(***********************************************************************************************)
(* HMI Alarme*)
(***********************************************************************************************)
FOR idx := 1 TO 500 BY 1 DO
    HMI.xArAlarmHMI[idx] := HMI.strArALARM[idx].xAlarmOUT;
END_FOR

FOR idx := 1 TO 100 BY 1 DO
    HMI.xArAlarmHMI[idx + 5000] := HMI.strArMSG[idx].xAlarmOUT;
END_FOR

(***********************************************************************************************)
(* Cycle Time *)
(***********************************************************************************************)
_FB_SystemTime(timeLoDW => dw_ActTime, timeHiDW =>);
dw_ActTime := dw_ActTime AND 16#FFFF0000;

IF HMI.btArMain[8].rtrig THEN
    HMI.PieceDoneTmp := 0;
END_IF

(***********************************************************************************************)
(* Operating hours  *)
(***********************************************************************************************)
(* 0.5' Blinker *)
BLINK_500(IN := NOT BLINK_500_.Q, PT := T#500MS, Q => x_BLINK_500);
BLINK_500_(IN := NOT BLINK_500.Q, PT := T#500MS);
(* 0.1' Blinker *)
BLINK_100(IN := NOT BLINK_100_.Q, PT := T#100MS, Q => x_BLINK_100);
BLINK_100_(IN := NOT BLINK_100.Q, PT := T#100MS);
(* 6' Ticker *)
TICK6M(IN := NOT TICK6M_.Q, PT := T#1MS, Q => x_TICK6M);
TICK6M_(IN := NOT TICK6M.Q, PT := t#6m);

(* Operating hours *)
IF TICK6M.Q THEN
    (* AUTO *)
    IF (HMI.enState = enState.StateAUTO) THEN
        PERS.udiCount6Mauto := PERS.udiCount6Mauto + 1;
        IF (PERS.udiCount6Mauto >= 10) THEN
            PERS.udiCount6Mauto := 0;
            PERS.udiCountHauto  := PERS.udiCountHauto + 1;
            IF (PERS.udiCountHauto < 0) THEN
                PERS.udiCountHauto := 0;
            END_IF;
        END_IF;
    END_IF;

    (* TOTAL *)
    PERS.udiCount6Mon := PERS.udiCount6Mon + 1;
    IF (PERS.udiCount6Mon >= 10) THEN
        PERS.udiCount6Mon := 0;
        PERS.udiCountHon  := PERS.udiCountHon + 1;
        IF (PERS.udiCountHon < 0) THEN
            PERS.udiCountHon := 0;
        END_IF;
    END_IF;

    //6h
    iCount6h := iCount6h + 1;
END_IF;

//Alarmlog schreiben nach 6h oder bei NOT-AUS
//rtNOTAUS(CLK:=_02_SAFETY.xOUT_ESout);
IF (iCount6h >= 60) OR rtNOTAUS.Q THEN
    iCount6h        := 0;
    HMI.xWriteALlog := NOT HMI.xWriteALlog;
END_IF;

END_PROGRAM

// ---- POUs/10_HMI/_14_STATE.TcPOU
PROGRAM _14_STATE
(****************************************************************************)
//STATE PROGRAMM
//	- Control Buttons
//	- Status Anlage
//
//	05.09.2019/Dj
//
//	Version:
(****************************************************************************)
VAR
    fb_State  : FB_State; //Status der Maschine
    sStateDbg : STRING;   // enState but in string format

    //Control Buttons
    _FB_btAUTO          : FB_BUTTON;
    _FB_btSTEP          : FB_BUTTON;
    _FB_btEND           : FB_BUTTON;
    _FB_btMANU          : FB_BUTTON;
    _FB_btINIT          : FB_BUTTON;
    _FB_btSTOP          : FB_BUTTON;
    _FB_btLEER          : FB_BUTTON;
    _FB_btQUIT          : FB_BUTTON;
    _FB_btSTART         : FB_BUTTON;
    _FB_btRESET_COUNTER : FB_BUTTON;
END_VAR

//****************************************************************************
// 	CONTROL BUTTONS
//****************************************************************************
//	AUTO 
_FB_btAUTO(pbtIN  := ADR(HMI.btArMain[0]),
           xINdis := (HMI.enState < enState.StateREADY),
           xINon  := (HMI.enState = enState.StateAUTO),
           xINerr := FALSE);

//STEP
_FB_btSTEP(pbtIN  := ADR(HMI.btArMain[1]),
           xINdis := (HMI.enState < enState.StateREADY),
           xINon  := (HMI.enState = enState.StateSTEP),
           xINerr := FALSE);

//END
_FB_btEND(pbtIN  := ADR(HMI.btArMain[2]),
          xINdis := (HMI.enState < enState.StateREADY),
          xINon  := (HMI.enState = enState.StateEND),
          xINerr := FALSE);

//MANU
_FB_btMANU(pbtIN  := ADR(HMI.btArMain[3]),
           xINdis := (HMI.enState > enState.StateSTEP) OR
                     (HMI.enState = enState.StateALARM) OR
                     (HMI.enState < enState.StateAIRon),
           xINon  := (HMI.enState = enState.StateMANU),
           xINerr := FALSE);

//INIT
_FB_btINIT(pbtIN  := ADR(HMI.btArMain[4]),
           xINdis := (HMI.enState < enState.StateENGIZED),
           xINon  := (HMI.enState = enState.StateINIT),
           xINerr := FALSE);

//STOP
_FB_btSTOP(pbtIN  := ADR(HMI.btArMain[5]),
           xINdis := (HMI.enState < enState.StateENGIZED),
           xINon  := FALSE,
           xINerr := FALSE);

//LEERFAHREN
_FB_btLEER(pbtIN  := ADR(HMI.btArMain[6]),
           xINdis := FALSE,
           xINon  := FALSE,
           xINerr := FALSE);

//QUIT
_FB_btQUIT(pbtIN  := ADR(HMI.btArMain[7]),
           xINdis := FALSE,
           xINon  := FALSE,
           xINerr := HMI.xAlarm);

_FB_btRESET_COUNTER(pbtIN  := ADR(HMI.btArMain[8]),
                    xINdis := FALSE,
                    xINon  := HMI.btArMain[8].press,
                    xINerr := FALSE);

//START
_FB_btSTART(pbtIN  := ADR(HMI.btArMain[9]),
            xINdis := HMI.enState < enState.StateREADY,
            xINon  := HMI.btArMain[9].on,
            xINerr := FALSE);

//****************************************************************************
// 	STATE FB
//****************************************************************************
fb_State(xIN_AutoInit   := FALSE,
         xIN_DoRef      := FALSE,
         xIN_ENERGIE    := _02_SAFETY.xOUT_MonOut,
         xIN_AIR        := IN.I004_druckwachter_luftdruck_ok,
         xIN_EINRICHTEN := _02_SAFETY.xOUT_Einrichten,
         xIN_AUTO       := HMI.btArMain[0].rtrig,
         xIN_STEP       := HMI.btArMain[1].rtrig,
         xIN_CYCLE      := HMI.btArMain[2].rtrig,
         xIN_MANU       := HMI.btArMain[3].rtrig,
         xIN_INIT       := HMI.btArMain[4].rtrig,
         xIN_STOP       := HMI.btArMain[5].rtrig,
         xIN_LEER       := HMI.btArMain[6].rtrig,
         xIN_InitEND    := (GVL.st105_aut.xOUT_InitDone) AND
                           (GVL.st110_aut.xOUT_InitDone) AND
                           (GVL.st115_aut.xOUT_InitDone) AND
                           (GVL.st120_aut.xOUT_InitDone) AND
                           (GVL.st125_aut.xOUT_InitDone) AND
                           (GVL.st130_aut.xOUT_InitDone) AND
                           (GVL.st135_aut.xOUT_InitDone) AND
                           (GVL.st140_aut.xOUT_InitDone) AND
                           (GVL.st145_aut.xOUT_InitDone) AND
                           (GVL.st150_aut.xOUT_InitDone) AND
                           (GVL.st155_aut.xOUT_InitDone) AND
                           (GVL.st160_aut.xOUT_InitDone) AND
                           (GVL.st165_aut.xOUT_InitDone) AND
                           (GVL.st170_aut.xOUT_InitDone) AND
                           (GVL.st175_aut.xOUT_InitDone) AND
                           (GVL.st176_aut.xOUT_InitDone) AND
                           (GVL.st180_aut.xOUT_InitDone) AND
                           (GVL.st185_aut.xOUT_InitDone),
         xIN_ALARM := MAIN.MoverMan.xOUT_Error OR
                      ((GVL.st105_aut.xOUT_AlarmST) OR
                      (GVL.st110_aut.xOUT_AlarmST) OR
                      (GVL.st115_aut.xOUT_AlarmST) OR
                      (GVL.st120_aut.xOUT_AlarmST) OR
                      (GVL.st125_aut.xOUT_AlarmST) OR
                      (GVL.st128_aut.xOUT_AlarmST) OR
                      (GVL.st130_aut.xOUT_AlarmST) OR
                      (GVL.st135_aut.xOUT_AlarmST) OR
                      (GVL.st140_aut.xOUT_AlarmST) OR
                      (GVL.st145_aut.xOUT_AlarmST) OR
                      (GVL.st150_aut.xOUT_AlarmST) OR
                      (GVL.st155_aut.xOUT_AlarmST) OR
                      (GVL.st160_aut.xOUT_AlarmST) OR
                      (GVL.st165_aut.xOUT_AlarmST) OR
                      (GVL.st170_aut.xOUT_AlarmST) OR
                      (GVL.st175_aut.xOUT_AlarmST) OR
                      (GVL.st180_aut.xOUT_AlarmST) OR
                      (GVL.st185_aut.xOUT_AlarmST)) AND
                      (GVL.st105_aut.xOUT_ErrFlag OR GVL.st105_aut.xOUT_Wait) AND
                      (GVL.st110_aut.xOUT_ErrFlag OR GVL.st110_aut.xOUT_Wait) AND
                      (GVL.st115_aut.xOUT_ErrFlag OR GVL.st115_aut.xOUT_Wait) AND
                      (GVL.st120_aut.xOUT_ErrFlag OR GVL.st120_aut.xOUT_Wait) AND
                      (GVL.st125_aut.xOUT_ErrFlag OR GVL.st125_aut.xOUT_Wait) AND
                      // we ignore the state of ST128
                      (GVL.st130_aut.xOUT_ErrFlag OR GVL.st130_aut.xOUT_Wait) AND
                      (GVL.st135_aut.xOUT_ErrFlag OR GVL.st135_aut.xOUT_Wait) AND
                      // we ignore the state of ST140
                      (GVL.st145_aut.xOUT_ErrFlag OR GVL.st145_aut.xOUT_Wait) AND
                      (GVL.st150_aut.xOUT_ErrFlag OR GVL.st150_aut.xOUT_Wait) AND
                      (GVL.st155_aut.xOUT_ErrFlag OR GVL.st155_aut.xOUT_Wait) AND
                      (GVL.st160_aut.xOUT_ErrFlag OR GVL.st160_aut.xOUT_Wait) AND
                      (GVL.st165_aut.xOUT_ErrFlag OR GVL.st165_aut.xOUT_Wait) AND
                      (GVL.st170_aut.xOUT_ErrFlag OR GVL.st170_aut.xOUT_Wait) AND
                      (GVL.st175_aut.xOUT_ErrFlag OR GVL.st175_aut.xOUT_Wait) AND
                      (GVL.st180_aut.xOUT_ErrFlag OR GVL.st180_aut.xOUT_Wait) AND
                      (GVL.st185_aut.xOUT_ErrFlag OR GVL.st185_aut.xOUT_Wait),
         xIN_LastDone := (NOT (HMI.enState = enState.StateLEER) OR
                         (MAIN.MoverMan.xOUT_AllMoverEmpty AND GVL.st185_aut.xOUT_Done)) AND
                         GVL.st105_aut.xOUT_Wait AND
                         GVL.st110_aut.xOUT_Wait AND
                         GVL.st115_aut.xOUT_Wait AND
                         GVL.st120_aut.xOUT_Wait AND
                         GVL.st125_aut.xOUT_Wait AND
                         GVL.st128_aut.xOUT_Wait AND
                         GVL.st130_aut.xOUT_Wait AND
                         GVL.st135_aut.xOUT_Wait AND
                         GVL.st140_aut.xOUT_Wait AND
                         GVL.st145_aut.xOUT_Wait AND
                         GVL.st150_aut.xOUT_Wait AND
                         GVL.st155_aut.xOUT_Wait AND
                         GVL.st160_aut.xOUT_Wait AND
                         GVL.st165_aut.xOUT_Wait AND
                         GVL.st170_aut.xOUT_Wait AND
                         GVL.st175_aut.xOUT_Wait AND
                         GVL.st180_aut.xOUT_Wait AND
                         GVL.st185_aut.xOUT_Wait,
         xIN_WaitFBs := GVL.st105_aut.xOUT_Wait AND
                        GVL.st110_aut.xOUT_Wait AND
                        GVL.st115_aut.xOUT_Wait AND
                        GVL.st120_aut.xOUT_Wait AND
                        GVL.st125_aut.xOUT_Wait AND
                        GVL.st128_aut.xOUT_Wait AND
                        GVL.st130_aut.xOUT_Wait AND
                        GVL.st135_aut.xOUT_Wait AND
                        GVL.st140_aut.xOUT_Wait AND
                        GVL.st145_aut.xOUT_Wait AND
                        GVL.st150_aut.xOUT_Wait AND
                        GVL.st155_aut.xOUT_Wait AND
                        GVL.st160_aut.xOUT_Wait AND
                        GVL.st165_aut.xOUT_Wait AND
                        GVL.st170_aut.xOUT_Wait AND
                        GVL.st175_aut.xOUT_Wait AND
                        GVL.st180_aut.xOUT_Wait AND
                        GVL.st185_aut.xOUT_Wait,
         enINOUT_State := HMI.enState);

sStateDbg := TO_STRING(HMI.enState);

END_PROGRAM

// ---- POUs/20_AUTO/ST175/Trumpf/TruMark_SingleCmds.TcPOU
PROGRAM TruMark_SingleCmds
(*
	TRUMPF Laser Marking Systems
	============================
	created: 11.01.2019 Erik Haller
	
     +============+
     |SingleCmds  |
     +============+
          |
          v
       +--+------+
       |Input    |	 Interface
       |  -----  |   if_TruMark
       |Output   |
       |  -----  |
       +---------+
               ^
               |
    +==================+
    |TruMark_Ethercat  |
    +==================+
	
	Software Disclaimer:
	THIS SOFTWARE IS PROVIDED "AS IS" AND ANY EXPRESSED OR IMPLIED WARRANTIES, INCLUDING, BUT NOT LIMITED TO,
	THE IMPLIED WARRANTIES OF MERCHANTABILITY AND FITNESS FOR A PARTICULAR PURPOSE ARE DISCLAIMED. 
	IN NO EVENT SHALL THE REGENTS OR CONTRIBUTORS BE LIABLE FOR ANY DIRECT, INDIRECT, INCIDENTAL, SPECIAL, EXEMPLARY, 
	OR CONSEQUENTIAL DAMAGES (INCLUDING, BUT NOT LIMITED TO, PROCUREMENT OF SUBSTITUTE GOODS OR SERVICES; LOSS OF USE, DATA, OR PROFITS;
	OR BUSINESS INTERRUPTION) HOWEVER CAUSED AND ON ANY THEORY OF LIABILITY, WHETHER IN CONTRACT, STRICT LIABILITY, OR TORT (INCLUDING NEGLIGENCE OR OTHERWISE) 
	ARISING IN ANY WAY OUT OF THE USE OF THIS SOFTWARE, EVEN IF ADVISED OF THE POSSIBILITY OF SUCH DAMAGE.
*)



VAR
	iStep : INT;
	abB1 : ARRAY [0..7] OF BOOL;	// used for TLV request 20261
	abB2 : ARRAY [0..7] OF BOOL;	// used for TLV request 20261
	iBitNo : INT;
	sFileName : STRING;
	sVar : STRING;
END_VAR

IF if_TruMark.bError THEN
	iStep := 0;
END_IF

CASE iStep OF
	0: 		// Initialisation
		IF NOT if_TruMark.bError AND NOT if_TruMark.bBusy THEN
			if_SingleCmds.bReady := TRUE;
			iStep := 5;
		END_IF
	
	5:		
		// ---------------------------------------------------------
		// TruMark_Ethercat is Ready --> SELECT Step-No
		// ---------------------------------------------------------
		
		IF if_SingleCmds.bStart THEN
			if_SingleCmds.bStart := FALSE;
			if_SingleCmds.bReady := FALSE;
			iStep := if_SingleCmds.iStepNr;
		END_IF
	
// ============================================================================================================================
// 			T L V   C O M M A N D S		iStep: 10 - 100
// ============================================================================================================================
		
	10:		// -----------------------------------------------------------
			// TLV - Activate Laser / Open Shutter				Attention! Not all Marking Laser have a Shutter
			// -----------------------------------------------------------
		IF NOT if_TruMark.bBusy THEN
			if_TruMark.diTlvTag := 20201;
			if_TruMark.sTlvValueIn := '1';
			if_TruMark.bTlvCmd := TRUE;	
		ELSE
			iStep := 11;
		END_IF
	11:		// Wait for response
		IF NOT if_TruMark.bBusy AND if_TruMark.Status.b0_Laser_On (*AND if_TruMark.Status.b1_Laser_Ready AND if_TruMark.Status.b3_Shutter_Open *) THEN
			iStep := 0;
		END_IF
		
	12:		// -----------------------------------------------------------
			// TLV - Deactivate Laser / Close Shutter				Attention! Not all Marking Laser have a Shutter
			// -----------------------------------------------------------
		IF NOT if_TruMark.bBusy THEN
			if_TruMark.diTlvTag := 20201;
			if_TruMark.sTlvValueIn := '0';
			if_TruMark.bTlvCmd := TRUE;
		ELSE
			iStep := 13;
		END_IF
	13:		// Wait for response
		IF NOT if_TruMark.bBusy AND NOT if_TruMark.Status.b0_Laser_On AND NOT if_TruMark.Status.b1_Laser_Ready (* AND NOT if_TruMark.Status.b3_Shutter_Open *) THEN
			iStep := 0;
		END_IF
				
	20:		// -----------------------------------------------------------
			// TLV - Load Marking File
			// -----------------------------------------------------------
		IF NOT if_TruMark.bBusy THEN
			if_TruMark.diTlvTag := 20401;
			if_TruMark.sTlvValueIn := if_SingleCmds.sInputValue;
			if_TruMark.bTlvCmd := TRUE;	
		ELSE
			iStep := 21;
		END_IF
	21:		// Wait for response
			// Default settings: Convert at start marking - Option: Convert at load marking file
			// 					TruTops Mark application: Extras -> 7 Konfiguration -> Verschiedenes [Zeitpunkt der Konvertierung]
		IF NOT if_TruMark.bBusy AND NOT if_TruMark.bError AND NOT if_TruMark.Status.b16_Conversion_Active THEN
			sFileName := if_SingleCmds.sInputValue;
			iStep := 0;
		END_IF

	30:		// -----------------------------------------------------------
			// TLV - Request state of conversion
			// -----------------------------------------------------------
		IF NOT if_TruMark.bBusy THEN
			if_TruMark.diTlvTag := 20222;
			if_TruMark.sTlvValueIn := '';
			if_TruMark.bTlvCmd := TRUE;
		ELSE
			iStep := 31;
		END_IF
	31:		// Wait for response
		// Option a). check TLV response
		IF NOT if_TruMark.bBusy AND NOT if_TruMark.bError THEN
			IF SIZEOF(if_TruMark.sTlvRespons) = 4 THEN			// The expected response has 4 bytes - 0x30, 0x00, [0x30 or 0x31], 0x00
				IF if_TruMark.sTlvRespons[2] = 16#30 THEN  
					iStep := 0;			// ASCII code 0x30 = '0' --> conversion is not active
				ELSE
					iStep := 30;		// ASCII code 0x31 = '1' --> conversion is active
										// Loop with TLV-Request and check on TLV-Response
				END_IF
			END_IF
		END_IF
		
		// Option b). check BIT-Status of bit 16
		IF NOT if_TruMark.bBusy AND NOT if_TruMark.bError AND NOT if_TruMark.status.b16_Conversion_Active THEN
			iStep := 0;
		END_IF

	35:		// -----------------------------------------------------------
			// TLV - Set Variable
			// -----------------------------------------------------------
		IF NOT if_TruMark.bBusy THEN
			if_TruMark.diTlvTag := 20421;
			if_TruMark.sTlvValueIn := if_SingleCmds.sInputValue;
			if_TruMark.bTlvCmd := TRUE;	
		ELSE
			iStep := 36;
		END_IF
	36:		// Wait for response
		IF NOT if_TruMark.bBusy AND NOT if_TruMark.bError THEN
			sVar := if_SingleCmds.sInputValue;
			iStep := 0;
		END_IF

	40:		// -----------------------------------------------------------
			// TLV - Request Laser state
			// -----------------------------------------------------------
		IF NOT if_TruMark.bBusy THEN
			if_TruMark.diTlvTag := 20261;
			if_TruMark.sTlvValueIn := '';
			if_TruMark.bTlvCmd := TRUE;
		ELSE
			iStep := 41;
		END_IF
	41:		// Wait for response
		IF NOT if_TruMark.bBusy AND NOT if_TruMark.bError THEN
			IF LEN(if_TruMark.sTlvRespons) = 20 THEN		// The expected response has 20 bytes
															// BitNo			0  1  2  3  4  5  6  7  8  9  10 11 12 13 14 15 16 17 18 19
															// TLV-Resp HEX:	30 00 30 30 30 30 31 31 31 31 00 30 30 30 31 31 30 30 30 00
															// TLV-Resp 		0  ;  0  0  0  0  1  1  1  1  ;  0  0  0  1  1  0  0  0  ;
															// Desc.			rc    B1                         B2	
				FOR iBitNo := 0 TO 7 BY 1 DO
					abB1[7-iBitNo] := if_TruMark.sTlvRespons[iBitNo+2] = 16#31;		// ASCII Code 0x31 = '1'
					abB2[7-iBitNo] := if_TruMark.sTlvRespons[iBitNo+11] = 16#31;
				END_FOR
				
				// Set your conditions	--> e.g. B1-Bit 7-0=00011111 / B2-Bit 15-8=01011011
				(*
					B1 [7-0]:
					Bit 7: 1	Laser hat eine Störung
					Bit 6: 1	Überwachung Laser hat angesprochen
					Bit 5: 0	Laser stabil (Diodenstrom im Band)
					Bit 4: 1	Strahlaufweiter in Position
					Bit 3: 1	Verschluss ist offen
					Bit 2: 1	Sicherheitskreis ist geschlossen
					Bit 1: 1	Laser ist bereit
					Bit 0: 1	Strahlquelle ist Ein
					
					B2 [15–8]:
					Bit 15: 1	Steuerung ist ein
					Bit 14: 1	Heizphase Laser ist ein
					Bit 13: 1	Not-Aus-Kreis ist geschlossen
					Bit 12: 1	Schlüsselschalter Lasersperre ist geschlossen.
					Bit 11: 1	Steuerung selbst ausschalten aktiviert
					Bit 10: 1	Q-Switch Trigger ist ein
					Bit 9:  1	Laserwarnlampe ist ein
					Bit 8:  1	Pilotlaser ist ein
				*)
				(* Original IF      abB1[0] AND abB1[1] AND     abB1[2] AND NOT abB1[3] AND abB1[4] AND abB1[5] AND NOT abB1[6] AND NOT abB1[7]
				AND NOT abB2[0] AND abB2[1] AND NOT abB2[2] AND NOT abB2[3] AND abB2[4] AND abB2[5] AND NOT abB2[6] AND     abB2[7] 
				*)
				IF      abB1[0] (* AND abB1[1] AND abB1[2] AND abB1[3] *)AND abB1[4] AND abB1[5] AND NOT abB1[6] AND NOT abB1[7]
				AND NOT abB2[0] AND abB2[1] AND NOT abB2[2] AND NOT abB2[3] AND abB2[4] AND abB2[5] AND NOT abB2[6] AND     abB2[7] 
				THEN  
					iStep := 0;
				ELSE
					// Conditions not matched
					iStep := 40;
				END_IF
				
				// We may be blocked for nothing, so we retry the command
			ELSIF NOT if_TruMark.bTlvCmd THEN
					iStep := 40;
			END_IF
		END_IF

	50:		// -----------------------------------------------------------
			// TLV - Start marking
			// -----------------------------------------------------------
		IF NOT if_TruMark.bBusy THEN
			if_TruMark.diTlvTag := 20204;
			if_TruMark.sTlvValueIn := '';
			if_TruMark.bTlvCmd := TRUE;
		ELSE
			iStep := 51;
		END_IF
	51:		// Wait for response
		IF NOT if_TruMark.bBusy THEN
			IF NOT if_TruMark.bError THEN
				IF NOT if_TruMark.Status.b15_Mark_Active THEN
					iStep := 0;	
				END_IF
			ELSE
				// Error
			END_IF
		END_IF

	55:		// -----------------------------------------------------------
			// TLV - Convert marking file
			// -----------------------------------------------------------
		IF NOT if_TruMark.bBusy THEN
			if_TruMark.diTlvTag := 20402;
			if_TruMark.sTlvValueIn := '';
			if_TruMark.bTlvCmd := TRUE;	
		ELSE
			iStep := 56;
		END_IF
	56:		// Wait for response
		IF NOT if_TruMark.bBusy AND NOT if_TruMark.bError THEN
			iStep := 0;
		END_IF		

// ============================================================================================================================
// 			B I T   C O M M A N D S		iStep: 100 - 200
// ============================================================================================================================
		
	100:	// -------------------------------------------------------
			// BIT 0 - Activate Laser / Open Shutter				Attention! Not all Marking Laser have a Shutter
			// -------------------------------------------------------
		if_TruMark.dwBitIn.0 := TRUE;
		if_TruMark.bBitCmd := TRUE;	
		iStep := 101;
	101:	// Wait for response
		IF NOT if_TruMark.bBusy AND if_TruMark.Status.b0_Laser_On AND if_TruMark.Status.b1_Laser_Ready (* AND if_TruMark.Status.b3_Shutter_Open *) THEN
			iStep := 0;
		END_IF
		
	102:	// -------------------------------------------------------
			// BIT 0 - Deactivate Laser / Close Shutter
			// -------------------------------------------------------
		if_TruMark.dwBitIn.0 := FALSE;
		if_TruMark.bBitCmd := TRUE;
		iStep := 103;
	103:	// Wait for response
		IF  NOT if_TruMark.bBusy AND NOT if_TruMark.Status.b0_Laser_On AND NOT if_TruMark.Status.b1_Laser_Ready (* AND NOT if_TruMark.Status.b3_Shutter_Open *) THEN
			iStep := 0;
		END_IF

	110:	// -------------------------------------------------------
			// BIT 1 - Open Shutter		Attention! Not all Marking Laser have a Shutter
			// -------------------------------------------------------
		if_TruMark.dwBitIn.1 := TRUE;
		if_TruMark.bBitCmd := TRUE;
		iStep := 111;
	111:	// Wait for response
		IF NOT if_TruMark.bBusy AND if_TruMark.Status.b3_Shutter_Open THEN
			iStep := 0;
		END_IF
		
	112:	// -------------------------------------------------------
			// BIT 1 - Close Shutter
			// -------------------------------------------------------
		if_TruMark.dwBitIn.1 := FALSE;
		if_TruMark.bBitCmd := TRUE;
		iStep := 113;
	113:	// Wait for response
		IF NOT if_TruMark.bBusy AND NOT if_TruMark.Status.b3_Shutter_Open THEN
			iStep := 0;
		END_IF

	120:	// -------------------------------------------------------
			// BIT 2 - Laser Reset
			// -------------------------------------------------------
		if_TruMark.dwBitIn.2 := TRUE;
		if_TruMark.bBitCmd := TRUE;
		iStep := 121;
	121:	// Wait for response
		IF NOT if_TruMark.bBusy (*dj2101 AND if_TruMark.Status.b0_Laser_On AND if_TruMark.Status.b1_Laser_Ready*) THEN
			if_TruMark.dwBitIn.2 := FALSE; 	// deactivate reset function
			if_TruMark.bBitCmd := TRUE;	
			iStep := 0;
		END_IF

	130:	// -------------------------------------------------------
			// BIT 3 - Pilot Laser On
			// -------------------------------------------------------
		if_TruMark.dwBitIn.3 := TRUE;
		if_TruMark.bBitCmd := TRUE;
		iStep := 131;
	131:	// Wait for response
		IF NOT if_TruMark.bBusy AND if_TruMark.Status.b7_PilotLaser_On THEN
			iStep := 0;
		END_IF
		
	132:	// -------------------------------------------------------
			// BIT 3 - Pilot Laser OFF
			// -------------------------------------------------------
		if_TruMark.dwBitIn.3 := FALSE;
		if_TruMark.bBitCmd := TRUE;
		iStep := 133;
	133:	// Wait for response
		IF NOT if_TruMark.bBusy AND NOT if_TruMark.Status.b7_PilotLaser_On THEN
			iStep := 0;
		END_IF
		
	180:	// -------------------------------------------------------
			// BIT 8 - Cancel Marking Process
			// -------------------------------------------------------
		if_TruMark.dwBitIn.8 := TRUE;
		if_TruMark.bBitCmd := TRUE;
		iStep := 181;
	181:	// Wait for response
		IF NOT if_TruMark.bBusy AND NOT if_TruMark.Status.b15_Mark_Active THEN
			iStep := 0;
		END_IF

END_CASE

END_PROGRAM

// ---- POUs/20_AUTO/ST105/FB_AUT_105.TcPOU
FUNCTION_BLOCK FB_AUT_105 EXTENDS FB_AUT_ABSTRACT
(****************************************************************************)
(*	POU_AUT_zxx			Bausteinaufrufe Station	zxx							*)
(*	Status				ungetestet											*)
(*  Version:			1.0													*)
(*	Beschrieb:																*)
(*																			*)
(*	Abläufe:			FB_ABLzxxA		Hauptablauf							*)
(*																			*)
(*																			*)
(* 	25.09.2019/Dj															*)
(****************************************************************************)
(*	dd.mm.yyyy   KZ    x.y			Beschrieb								*)
(****************************************************************************)
VAR_INPUT
    (* spezifische Eingänge *)

END_VAR
VAR_OUTPUT
    (* spezifische Ausgänge *)

END_VAR
VAR
    (* Bausteine *)
    fb_Pnp    : FB_ABL_105_Pnp;
    fb_Feeder : FB_ABL_105_Feeder;

    fb_stat_pnp    : FB_AUT_Statistics;
    fb_stat_Feeder : FB_AUT_Statistics;
END_VAR

VAR CONSTANT
END_VAR

(*******************************************************************)
(* Timer *)
(*******************************************************************)

(*******************************************************************)
(* Flanken / Merker *)
(*******************************************************************)
//MANU CYCLE
IF (enIN_State = StateMANU) AND xIN_ManuCycle THEN
    xManuCycle := TRUE;
END_IF;

IF (enIN_State <> StateMANU) OR xOUT_Done THEN
    xManuCycle := FALSE;
END_IF

//NEXT STEP
xNextStep := (enIN_State > StateSTEP) OR
             ((enIN_State = StateSTEP) AND xIN_Step) OR
             ((enIN_State = StateMANU) AND xManuCycle);

//RESET
xReset := (enIN_State < StateREADY) AND (enIN_State <> StateINIT) AND NOT xManuCycle;

(*******************************************************************)
(* Bausteinaufrufe Abläufe *)
(*******************************************************************)

xRelease := MAIN.MoverMan.IsProcessUsed(THIS^);

fb_Pnp(xIN_Reset       := xReset,
       xIN_Init        := xIN_Init,
       xIN_Quit        := xIN_Quit,
       xIN_Start       := enIN_State >= enState.StateLEER AND xRelease,
       xIN_Sperre      := NOT xIN_On,
       xIN_NextStep    := xNextStep,
       xIN_AlarmAktiv  := xIN_AlarmAktiv,
       xIN_DryCycle    := xIN_DryCycle,
       xIN_RestartCYCL := enIN_State >= enState.StateLEER, //            
       enIN_State      := enIN_State,
       tIN_Timeout     := tIN_Timeout,
       pxFG_Freigabe   := ADR(xRelease),
       // special
       Mover              := THIS^.Mover,
       xIN_PceReadyToPick := fb_Feeder.xOUT_PceReadyToPick);

fb_Feeder(xIN_Reset       := xReset,
          xIN_Init        := xIN_Init,
          xIN_Quit        := xIN_Quit,
          xIN_Start       := enIN_State = enState.StateAUTO AND xRelease,
          xIN_Sperre      := NOT xIN_On,
          xIN_NextStep    := xNextStep,
          xIN_AlarmAktiv  := xIN_AlarmAktiv,
          xIN_DryCycle    := xIN_DryCycle,
          xIN_RestartCYCL := enIN_State = enState.StateAUTO,
          enIN_State      := enIN_State,
          tIN_Timeout     := tIN_Timeout,
          pxFG_Freigabe   := ADR(xRelease),
          // special
          xIN_PickPiece            := fb_Pnp.xOUT_PickPiece,
          xIN_RotTableBlockedByPnp := fb_Pnp.iOUT_Step = ST105_Pnp_e.Robot_wait_picked_falling OR
                                      fb_Pnp.iOUT_Step = ST105_Pnp_e.Robot_Pick OR
                                      fb_Pnp.iOUT_Step = ST105_Pnp_e.pusher_down OR
                                      fb_Pnp.iOUT_Step = ST105_Pnp_e.Init_HomeVertical OR
                                      fb_Pnp.iOUT_Step = ST105_Pnp_e.Init_VerticalDown);

fb_stat_pnp(xIN_Enable  := enState.StateAUTO = enIN_State,
            xIN_Waiting := fb_Pnp.xOUT_Wait,
            xIN_Running := (fb_Pnp.iOUT_Step >= ST105_Pnp_e.START) AND
                           (fb_Pnp.iOUT_Step <= ST105_Pnp_e.DONE),
            // Since we use a mover system, a cycle is done when we are waiting on a mover
            xIN_Done := fb_Pnp.iOUT_Step = ST105_Pnp_e.waitOnMover);

fb_stat_Feeder(xIN_Enable  := enState.StateAUTO = enIN_State,
               xIN_Waiting := fb_feeder.xOUT_Wait,
               xIN_Running := (fb_feeder.iOUT_Step >= ST105_Feeder_e.START) AND
                              (fb_feeder.iOUT_Step <= ST105_Feeder_e.DONE),
               xIN_Done := fb_feeder.iOUT_Step = ST105_Feeder_e.DONE);

(*******************************************************************)
(* Mover reset flags *)
(*******************************************************************)

(*******************************************************************)
(* OUTPUT *)
(*******************************************************************)
xOUT_InitDone := fb_Pnp.xOUT_InitDone AND fb_Feeder.xOUT_InitDone;
xOUT_Ready    := fb_Pnp.xOUT_Ready AND fb_Feeder.xOUT_Ready;
xOUT_Done     := fb_Pnp.xOUT_Done AND fb_Feeder.xOUT_Done;
xOUT_ErrFlag  := fb_Pnp.xOUT_ErrFlag OR fb_Feeder.xOUT_ErrFlag;
xOUT_Wait     := fb_Pnp.xOUT_Wait; // We don't wait on the feeder part here, too slow
xOUT_AlarmST  := xOUT_ErrFlag;

(*******************************************************************)
(* Bausteinaufruf Error Station *)
(*******************************************************************)
// POU_ERR_VORLAGE(xIN_QUIT:=xIN_Quit , pstrArIN_ALARM:=ADR(HMI.strArALARM[1]));

(* % of completion of the process *)
PROPERTY iCompletionPC : INT
GET
iCompletionPC := THIS^.fb_Pnp.iOUT_ProcessCompletion;
END_GET
END_PROPERTY

PROPERTY ProcessExecution : ProcessExecution_e
GET
ProcessExecution := THIS^._ProcessExecution;
END_GET
SET
THIS^._ProcessExecution := ProcessExecution;
END_SET
END_PROPERTY

PROPERTY xBusy : BOOL
GET
xBusy := THIS^.fb_Pnp.xOUT_Busy;
END_GET
SET
END_SET
END_PROPERTY

PROPERTY xDone : BOOL
GET
xDone := THIS^.fb_Pnp.xOUT_Ready OR THIS^.fb_Pnp.xOUT_Done;
END_GET
END_PROPERTY

PROPERTY xMoverPathFree : BOOL
GET
xMoverPathFree := THIS^.fb_Pnp.xOUT_MoverFree OR THIS^.fb_Pnp.xOUT_Ready OR THIS^.fb_Pnp.xOUT_Done;
END_GET
END_PROPERTY

PROPERTY xMoverShouldLeave : BOOL
GET
xMoverShouldLeave := THIS^.fb_Pnp.iOUT_Step = ST105_Pnp_e.SYNC_MOVER_LEAVE;
END_GET
END_PROPERTY

END_FUNCTION_BLOCK

// ---- POUs/20_AUTO/ST105/FB_ABL_105_Pnp.TcPOU
FUNCTION_BLOCK FB_ABL_105_Pnp
(****************************************************************************************)
(*	TITEL				RFID-Ring laden		    										*)
(*	Status				ungetestet                         								*)
(*	Beschrieb:			Ablaufbeschreibung												*)
(*																						*)
(*	Steps:	self-explained using enum													*)
(***********************************Revisionen*******************************************)
(*	see github blames																	*)
(****************************************************************************************)

VAR_INPUT
    xIN_Reset       : BOOL;          // Schrittkette zurücksetzen 
    xIN_Init        : BOOL;          // Initialisieren
    xIN_Quit        : BOOL;          // Fehler quittieren 
    xIN_Start       : BOOL;          // Startbefehl
    xIN_Sperre      : BOOL;          // FB Sperren 
    xIN_NextStep    : BOOL;          // Nächsten Schritt ausführen 
    xIN_AlarmAktiv  : BOOL;          // Anlage hat Alarm
    xIN_DryCycle    : BOOL;          // Fahren ohne Teile
    xIN_RestartCYCL : BOOL;          // Zyklus erneut starten im STEP, END, LEERFAHREN
    enIN_State      : enState;       // Status Anlage
    tIN_Timeout     : TIME := T#10s; // Timout

    pxFG_Freigabe : POINTER TO BOOL; //Freigabe von Station

    // Application specific
    Mover              : REFERENCE TO FB_Mover;
    xIN_PceReadyToPick : BOOL; // the piece(s) is/are ready to picked
END_VAR
VAR_OUTPUT
    (* standart Ausgänge *)
    xOUT_ErrFlag  : BOOL;        // Error Flag 
    xOUT_Busy     : BOOL;        // Baustein befindet sich im Ablauf 
    xOUT_Done     : BOOL;        // Baustein hat den Ablauf beendet 		
    xOUT_Ready    : BOOL;        // Ready to begin, should be the same state as done	
    xOUT_Timeout  : BOOL;        // Timeout FB 
    xOUT_InitDone : BOOL;        // initialisierung fertig
    xOUT_Wait     : BOOL;        // Wartet auf Bedingung
    iOUT_Step     : ST105_Pnp_e; // Aktueller Schritt 
    sOUT_Step     : STRING;      // Aktueller Schritt but in string format
    bOUT_Error    : BYTE;        // Fehlernummer

    iOUT_ProcessCompletion : INT;  //process completion, express in % (0-100)
    xOUT_MoverFree         : BOOL; // The mover is free to move
    xOUT_PickPiece         : BOOL; // Set to true when a piece is picked

END_VAR
VAR
    (* Standard *)
    (* Schritt *)
    iLastStep : ST105_Pnp_e; // Merker letzter Schritt 
    iPreStep  : ST105_Pnp_e; // Schritt zurück nach Alarm 
    iAktStep  : ST105_Pnp_e; // aktueller Schritt

    // Trigger Starten 
    rtSTART : R_TRIG;
    // Timer TimeOut 
    TON_Timeout : TON;

    (* Bausteine *)

    (* Spezial *)
    fb_axis105_11Z : FB_AxisLM_V1_1;

    fb_PnpVerAxisU : FB_LinearMotionMan;

    fb_simu_axis105_11Z : FB_Simu_AxisLM_V1_1;

    fanuc_cmd    AT %Q* : Fanuc_hw_command_to_robot_t;
    fanuc_status AT %I* : Fanuc_status_std_from_robot;

    aut_cmd_to_robot      AT %Q* : ST105_Fanuc_command_t;
    aut_status_from_robot AT %I* : ST105_Fanuc_status_t;

    PickOffset_X_deci AT %Q* : UINT; // X offset of picking position
    PickOffset_Y_deci AT %Q* : UINT; // Y offset of picking position
    PickUpPos_Z_deci  AT %Q* : UINT; // Z traveling height from pick to place position

    hmi_force_place    : BOOL;
    hmi_force_in_place : BOOL;

END_VAR
VAR CONSTANT
    PNP_SIMULATION : BOOL := FALSE; // Set to TRUE to simulate this part of the program
END_VAR

(*******************************************************************)
(* Trigger  *)
(*******************************************************************)
(* Zurücksetzen *)
IF xIN_RESET THEN
    iPreStep  := ST105_Pnp_e.RESET;
    iOUT_Step := ST105_Pnp_e.RESET;
END_IF;

(* Error Quittieren *)
IF (bOUT_Error <> 0) AND xIN_Quit THEN
    xOUT_ErrFlag := FALSE;
    bOUT_Error   := 0;
    iOUT_Step    := iPreStep;
END_IF;

(*******************************************************************)
(* Timer *)
(*******************************************************************)
TON_Timeout(IN := xIN_NextStep AND (iLastStep = iOUT_Step) (*todo FG *) ,
            PT := tIN_Timeout);

(*******************************************************************)
(* Bausteine *)
(*******************************************************************)
fb_PnpVerAxisU(config          := _20_AUTO.recipe.linearAxis[LinearAxis_e.ST105_11Z],
               xIN_Init        := enIN_State = enState.StateINIT,
               xIN_Reset       := xIN_Reset,
               lrIN_CurrPos    := fb_axis105_11Z.rOUT_ActPos,
               lrIN_Delta_mm   := 0.5,
               iIN_CurrentStep := iOUT_Step,
               iIN_moveNumber  := ST105_PnpVerPushPos_e._max);

fb_simu_axis105_11Z(xIN_Enable          := PNP_SIMULATION AND CONST.USE_SIMULATION,
                    bIN_AxisCntr        := fb_axis105_11Z.bOUT_AxisCntr,
                    wIN_AxisState       := ST105_Axis.axis105_11Z.wState,
                    udiIN_HomingTime_ms := 2000,
                    pIN_axisSimu        := ADR(SIMU.axis_ref[Axis_e.ST105_11Z]),
                    pIN_axisHW          := ADR(ST105_Axis.axis105_11Z.axis),
                    rIN_PosActual       := ST105_Axis.axis105_11Z.rActPos,
                    rIN_PosMax          := ST105_Axis.const105_11Z.POS_MAX,
                    rIN_PosMin          := ST105_Axis.const105_11Z.POS_MIN,
                    rIN_PixMax          := 100,
                    rIN_PixMin          := 0);

fb_axis105_11Z(enIN_State       := enIN_State,
               parIN_Buttons    := ADR(AXIS.btTeachArAxis[Axis_e.ST105_11Z]),
               xIN_DisButtons   := FALSE,
               xIN_Quit         := xIN_Quit,
               xIN_PARAMok      := TRUE,
               xIN_FREE         := TRUE,
               xIN_FREE_HOME    := TRUE,
               rIN_POSMIN       := ST185_Axis.const185_10Z.POS_MIN,
               rIN_POSMAX       := ST185_Axis.const185_10Z.POS_MAX,
               rIN_VELOMAX      := ST185_Axis.const185_10Z.VELO_MAX,
               rIN_VELOMANU     := ST185_Axis.const185_10Z.VELO_MANU,
               rIN_VELOOPEN     := ST185_Axis.const185_10Z.POS_MAX / 4,
               rIN_JogInc       := AXIS.rTeachIncAxis,
               xIN_Execute      := fb_PnpVerAxisU.xOUT_Execute,
               xIN_Relative     :=,
               xIN_STOP         :=,
               xIN_OFF          :=,
               rIN_Position     := TO_REAL(fb_PnpVerAxisU.OUT_MoveProfile.lrPosition),
               rIN_Velocity     := TO_REAL(fb_PnpVerAxisU.OUT_MoveProfile.lrVelocity),
               rIN_Acceleration := TO_REAL(fb_PnpVerAxisU.OUT_MoveProfile.lrAccel),
               rIN_Deceleration := TO_REAL(fb_PnpVerAxisU.OUT_MoveProfile.lrDecel),
               rIN_Jerk         := TO_REAL(fb_PnpVerAxisU.OUT_MoveProfile.lrJerk),
               rIN_PosManu      := TO_REAL(_20_AUTO.recipe.linearAxis[LinearAxis_e.ST105_11Z]
                                               .movesList[AXIS.bTeachPos[Axis_e.ST105_11Z]].lrPosition),
               rIN_VeloJogManu := TO_REAL(Axis.rJogVelo_pc),
               xIN_Home        := ST105_Pnp_e.Init_HomeVertical = iOUT_Step,
               xIN_Reset       := (ST105_Pnp_e.RESET = iOUT_Step) OR xIN_Reset,
               wAxisState      := fb_simu_axis105_11Z.wOUT_AxisState,
               bOUT_AxisCntr   => ST105_Axis.axis105_11Z.bCtrlHi,
               rOUT_ActPos     => ST105_Axis.axis105_11Z.rActPos,
               axisIN_REF      := fb_simu_axis105_11Z.pOUT_axisRef^);

(*******************************************************************)
(* OUTPUTS *)
(*******************************************************************)
// Error Flag 
xOUT_ErrFlag := (bOUT_Error <> 0) OR (ST105_Pnp_e.ERROR = iOUT_Step);
// Baustein befindet sich im Ablauf 
xOUT_Busy := (iOUT_Step > ST105_Pnp_e.READY) AND (iOUT_Step < ST105_Pnp_e.DONE);
// Baustein hat den Ablauf beendet
xOUT_Done := (iOUT_Step = ST105_Pnp_e.DONE);
// Process ready
xOUT_Ready := (iOUT_Step = ST105_Pnp_e.READY) OR (iOUT_Step = ST105_Pnp_e.waitOnMover);
// Timeout FB 				 		
xOUT_Timeout := TON_Timeout.Q;
// Itialisierung fertig			
xOUT_InitDone := (iOUT_Step = ST105_Pnp_e.READY) OR (iOUT_Step = ST105_Pnp_e.waitOnMover);
// Aktueller Schritt			
iOUT_Step := iOUT_Step; //Im Ablauf gesetzt		
sOUT_Step := TO_STRING(iOUT_Step);
//Fehlernummer	 
bOUT_Error := bOUT_Error; //Im Ablauf/FB gesetzt	
(* Warte (alle Schritte wo auf FG oder Teile gewartet wird) *)
xOUT_Wait := (iOUT_Step = ST105_Pnp_e.DONE) OR
             (iOUT_Step = ST105_Pnp_e.READY) OR
             (iOUT_Step = ST105_Pnp_e.START) OR
             (iOUT_Step = ST105_Pnp_e.waitOnMover) OR
             (iOUT_Step = ST105_Pnp_e.SYNC_MOVER_LEAVE) OR
             (iOUT_Step = ST105_Pnp_e.wait_on_feeder);

xOUT_MoverFree := iOUT_Step >= ST105_Pnp_e.MOVER_FREE_OP AND iOUT_Step < ST105_Pnp_e.MOVER_NEEDED_OP;

iOUT_ProcessCompletion := F_GetPercent_2(iOUT_Step,
                                         ST105_Pnp_e.wait_on_feeder,
                                         ST105_Pnp_e.pusher_down,
                                         ST105_Pnp_e.Robot_place,
                                         ST105_Pnp_e.pusher_down);

xOUT_PickPiece := iOUT_Step = ST105_Pnp_e.pusher_down;

fanuc_cmd.command_std.IMDSTP     := TRUE AND NOT (PNP_SIMULATION AND CONST.USE_SIMULATION);
fanuc_cmd.command_std.Hold       := TRUE AND NOT (PNP_SIMULATION AND CONST.USE_SIMULATION);
fanuc_cmd.command_std.SFSPD      := TRUE AND NOT (PNP_SIMULATION AND CONST.USE_SIMULATION);
fanuc_cmd.command_std.FaultReset := xIN_Quit;
fanuc_cmd.command_std.Start      := iOUT_Step = ST105_Pnp_e.Init_RobotRaiseStartFlag AND
                                    NOT (PNP_SIMULATION AND CONST.USE_SIMULATION);

fanuc_cmd.command_std.Enable := TRUE AND NOT (PNP_SIMULATION AND CONST.USE_SIMULATION);

PickOffset_X_deci := _20_AUTO.recipe.st105.PickOffset_X_deci;
PickOffset_Y_deci := _20_AUTO.recipe.st105.PickOffset_Y_deci;
// add a constant to adjust the screw height of the rotative table
PickUpPos_Z_deci := _20_AUTO.recipe.st105.PickUpPos_Z_deci + UINT#500;

aut_cmd_to_robot.FG_Pick  := (ST105_Pnp_e.Robot_Pick = iOUT_Step) AND NOT (PNP_SIMULATION AND CONST.USE_SIMULATION);
aut_cmd_to_robot.FG_Place :=
    ((ST105_Pnp_e.Robot_place = iOUT_Step) OR hmi_force_place) AND NOT (PNP_SIMULATION AND CONST.USE_SIMULATION);

aut_cmd_to_robot.Use_griper_left  := _20_AUTO.recipe.st105.xUseVerLeft;
aut_cmd_to_robot.Use_griper_right := _20_AUTO.recipe.st105.xUseVerRight;

aut_cmd_to_robot.XOff := _20_AUTO.recipe.st105.isPickOffset_X_neg;
aut_cmd_to_robot.YOff := _20_AUTO.recipe.st105.isPickOffset_Y_neg;
aut_cmd_to_robot.ZOff := _20_AUTO.recipe.st105.isPickUpPos_Z_neg;

(*******************************************************************)
(* Ablauf *)
(*******************************************************************)

(* Sperren *)
IF xIN_Sperre THEN
    iPreStep  := ST105_Pnp_e.RESET;
    iOUT_Step := ST105_Pnp_e.RESET;
    RETURN;
END_IF;

(* Schritt Merker *)
IF iAktStep <> iOUT_Step THEN
    iLastStep := iAktStep;
    iAktStep  := iOUT_Step;
END_IF

(* START *)
rtSTART(CLK := xIN_Start);

(*******************************************************************)
(* Schrittkette  *)
(*******************************************************************)
CASE iOUT_Step OF

(***** RESET *****)
ST105_Pnp_e.RESET: (* Schritt 0-99 *)
    //Initialisierungen
    //Start Init Ablauf
    IF xIN_Init THEN
        iOUT_Step := ST105_Pnp_e.INIT;
        //Start Manu Ablauf
    ELSIF enIN_State = StateMANU AND xIN_NextStep THEN
        iOUT_Step := ST105_Pnp_e.INIT;
    END_IF;

(***** INIT *****)
ST105_Pnp_e.INIT: (* Grundstellung ? *)
    IF fb_axis105_11Z.xOUT_HOMED THEN
        iOUT_Step := ST105_Pnp_e.Init_VerticalDown;
    ELSE
        iOUT_Step := ST105_Pnp_e.Init_HomeVertical;
    END_IF

ST105_Pnp_e.Init_HomeVertical:
    IF fb_axis105_11Z.xOUT_HOMED THEN
        iOUT_Step := ST105_Pnp_e.Init_VerticalDown;
    END_IF

ST105_Pnp_e.Init_VerticalDown:
    IF fb_PnpVerAxisU.MoveTo(ST105_PnpVerPushPos_e.down).xOUT_InPos THEN
        IF fanuc_status.PRG_Running THEN
            iOUT_Step := ST105_Pnp_e.Init_check_if_pces_handled;
        ELSE
            iOUT_Step := ST105_Pnp_e.Init_RobotRaiseStartFlag;
        END_IF
    END_IF

ST105_Pnp_e.Init_RobotRaiseStartFlag:
    IF TRUE THEN // maybe a tempo or a flag from the robot is needed here
        iOUT_Step := ST105_Pnp_e.Init_check_if_pces_handled;
    END_IF

ST105_Pnp_e.Init_RobotFallStartFlag:
    IF fanuc_status.PRG_Running OR (PNP_SIMULATION AND CONST.USE_SIMULATION) THEN
        iOUT_Step := ST105_Pnp_e.Init_check_if_pces_handled;
    END_IF

ST105_Pnp_e.Init_check_if_pces_handled:
    IF TRUE THEN
        IF aut_status_from_robot.Ready_to_place THEN
            iOUT_Step := ST105_Pnp_e.waitOnMover;
        ELSE
            iOUT_Step := ST105_Pnp_e.READY;
        END_IF
    END_IF

(***** READY / INIT DONE *****)
ST105_Pnp_e.READY:    (* Start AUTO,END,LEER,STEP *)
    IF xIN_Start THEN //IF rtSTART.Q THEN
        iOUT_Step := ST105_Pnp_e.START;
    END_IF

(***** START  ZYKLISCH *****)
ST105_Pnp_e.START: (*  *)
    IF xIN_NextStep AND pxFG_Freigabe^ THEN
        IF enState.StateLEER = enIN_State THEN
            IF aut_status_from_robot.Ready_to_place THEN
                iOUT_Step := ST105_Pnp_e.waitOnMover;
            ELSIF __ISVALIDREF(Mover) THEN
                iOUT_Step := ST105_Pnp_e.SYNC_MOVER_LEAVE;
            END_IF
        ELSE
            iOUT_Step := ST105_Pnp_e.wait_on_feeder;
        END_IF
    END_IF;

ST105_Pnp_e.wait_on_feeder:
    IF xIN_NextStep AND xIN_PceReadyToPick THEN
        iOUT_Step := ST105_Pnp_e.push_up_casing;
    END_IF

ST105_Pnp_e.push_up_casing:
    IF xIN_NextStep AND fb_PnpVerAxisU.MoveTo(ST105_PnpVerPushPos_e.up).xOUT_InPos THEN
        IF PNP_SIMULATION AND CONST.USE_SIMULATION THEN
            IF fb_axis105_11Z.xOUT_DONE THEN // needed beacause we perform 2 movements one after the other
                iOUT_Step := ST105_Pnp_e.pusher_down;
            END_IF
        ELSE
            iOUT_Step := ST105_Pnp_e.Robot_Pick;
        END_IF
    END_IF

ST105_Pnp_e.Robot_Pick:
    IF aut_status_from_robot.Picked THEN
        iOUT_Step := ST105_Pnp_e.Robot_wait_picked_falling;

        // we don't generate an error here since this may hapen
        // when we stop the machine during the robot movement
    ELSIF aut_status_from_robot.Ready_to_place THEN
        iOUT_Step := ST105_Pnp_e.waitOnMover;

    END_IF

ST105_Pnp_e.Robot_wait_picked_falling:
    IF xIN_NextStep AND NOT aut_status_from_robot.Picked THEN
        iOUT_Step := ST105_Pnp_e.pusher_down;
    END_IF

ST105_Pnp_e.pusher_down:
    IF xIN_NextStep AND fb_PnpVerAxisU.MoveTo(ST105_PnpVerPushPos_e.down).xOUT_InPos THEN
        iOUT_Step := ST105_Pnp_e.waitOnMover;
    END_IF

ST105_Pnp_e.waitOnMover: (*  *)
    IF xIN_NextStep AND (__ISVALIDREF(Mover) OR HMI.bArForceCyclusState[StationList_e.ST105]) THEN
        IF (PNP_SIMULATION AND CONST.USE_SIMULATION) OR
           ((enState.StateLEER = enIN_State) AND NOT aut_status_from_robot.Ready_to_place) THEN
            iOUT_Step := ST105_Pnp_e.SYNC_MOVER_LEAVE;
        ELSE
            IF Mover.GetLastStationDone() >= INT#105 THEN
                iOUT_Step := ST105_Pnp_e.SYNC_MOVER_LEAVE;
            ELSE
                iOUT_Step := ST105_Pnp_e.Robot_place;
            END_IF
        END_IF
    END_IF;

ST105_Pnp_e.Robot_place:
    IF aut_status_from_robot.Placed THEN
        iOUT_Step := ST105_Pnp_e.Robot_wait_placed_falling;

        IF __ISVALIDREF(Mover) THEN
            IF NOT Mover.SetLastStation(-105) THEN
                ASSERT(0);
            END_IF
        END_IF

        // we don't generate an error here since this may hapen
        // when we stop the machine during the robot movement
    ELSIF aut_status_from_robot.Ready_to_pick THEN
        iOUT_Step := ST105_Pnp_e.wait_on_feeder;

    END_IF

ST105_Pnp_e.Robot_wait_placed_falling:
    IF xIN_NextStep AND NOT aut_status_from_robot.Placed THEN
        iOUT_Step := ST105_Pnp_e.SYNC_MOVER_LEAVE;

        IF __ISVALIDREF(Mover) THEN
            IF NOT Mover.SetLastStation(105) THEN
                ASSERT(0);
            END_IF
        END_IF
    END_IF

ST105_Pnp_e.SYNC_MOVER_LEAVE:
    // The mover needs to be taken by MoverMan
    IF NOT __ISVALIDREF(Mover) THEN
        IF NOT aut_status_from_robot.Ready_to_place THEN
            iOUT_Step := ST105_Pnp_e.DONE;
        ELSE
            iOUT_Step := ST105_Pnp_e.waitOnMover;
        END_IF
    END_IF

(***** DONE *****)
ST105_Pnp_e.DONE: (* Letzter Schritt  *)
    IF NOT xIN_AlarmAktiv THEN
        //AUTO
        IF (enIN_State = StateAUTO) AND xIN_RestartCYCL THEN
            iOUT_Step := ST105_Pnp_e.START;
            //STEP / END / LEERFAHREN restart
        ELSIF (enIN_State < StateAUTO) AND (enIN_State >= enState.StateSTEP) AND xIN_RestartCYCL THEN
            iOUT_Step := ST105_Pnp_e.START;
            //STEP / END / LEERFAHREN fertig
        ELSIF (enIN_State = StateREADY) THEN
            iOUT_Step := ST105_Pnp_e.READY;
        END_IF;
    END_IF;

(************ ERROR *************)
ST105_Pnp_e.ERROR: (* ERROR *) ;

END_CASE;

END_FUNCTION_BLOCK

// ---- POUs/20_AUTO/Simu/FB_Simu_AxisLM_V1_1.TcPOU
FUNCTION_BLOCK FB_Simu_AxisLM_V1_1
VAR_INPUT
    xIN_Enable          : BOOL;          // When true, this FB simulate output signals
    bIN_AxisCntr        : BYTE;          // Axis Controlword
    wIN_AxisState       : WORD;          // Statuswort input, copy to output when fb is not enable
    udiIN_HomingTime_ms : UDINT := 2000; // homing time, expressed as millisecond

    pIN_axisSimu : POINTER TO AXIS_REF; // simulation axis ref, without hardware connection
    pIN_axisHW   : POINTER TO AXIS_REF; // hardware axis ref, the one wich is connected to hardware

    rIN_PosActual : REAL;
    rIN_PosMax    : REAL;
    rIN_PosMin    : REAL;
    rIN_PixMax    : INT;
    rIN_PixMin    : INT;
END_VAR
VAR_OUTPUT
    wOUT_AxisState : WORD;                //Statuswort
    rOUT_PixActual : INT;                 // actual position of the axis in pixel
    pOUT_axisRef   : POINTER TO AXIS_REF; // current axis ref used
END_VAR
VAR
    _iStep                 : INT;   // current step
    _udiStartHomingTime_ms : UDINT; // start homing time in ms
END_VAR
VAR CONSTANT
END_VAR

IF xIN_Enable THEN
    CASE _iStep OF
    0: // GET Ctrl-Bit 
        wOUT_AxisState := 16#0;

        IF bIN_AxisCntr.3 THEN
            _iStep := 10;
        END_IF

    10: // SET Status Bit #8
        wOUT_AxisState.7       := TRUE;
        _udiStartHomingTime_ms := GetTick();
        _iStep                 := 20;

    20: // Perform homing
        IF (GetTick() - _udiStartHomingTime_ms) > udiIN_HomingTime_ms THEN
            wOUT_AxisState.7 := FALSE;
            _iStep           := 30;
        END_IF

    30: // GET Ctrl-bit
        IF NOT bIN_AxisCntr.3 THEN
            _iStep := 40;
        END_IF

    40: // Status Bit #13
        wOUT_AxisState.12 := TRUE;
        _iStep            := 50;

    50: // ready, wait homing signal
        IF bIN_AxisCntr.3 THEN
            _iStep := 0;
        END_IF

    END_CASE

    pOUT_axisRef := pIN_axisSimu;

ELSE
    wOUT_AxisState := wIN_AxisState;
    _iStep         := 0;
    pOUT_axisRef   := pIN_axisHW;
END_IF

rOUT_PixActual := MAP_REAL_TO_INT(rValue    := rIN_PosActual,
                                  rFromHigh := rIN_PosMax,
                                  rFromLow  := rIN_PosMin,
                                  rToHigh   := rIN_PixMax,
                                  rToLow    := rIN_PixMin);

END_FUNCTION_BLOCK

// ---- POUs/20_AUTO/TOOL/GetTick.TcPOU
FUNCTION GetTick : UDINT
VAR_INPUT
END_VAR
VAR
END_VAR

GetTick := TO_UDINT(F_GetTaskTime()/10000);

END_FUNCTION

// ---- POUs/20_AUTO/TOOL/MAP_REAL_TO_INT.TcPOU
// Map a value from a given range in REAL inside a given range in INT format
// more about the MAP function here :
// https://www.arduino.cc/reference/en/language/functions/math/map/
FUNCTION MAP_REAL_TO_INT : INT
VAR_INPUT
    rValue    : REAL;
    rFromLow  : REAL;
    rFromHigh : REAL;
    rToLow    : INT;
    rToHigh   : INT;
END_VAR
VAR
END_VAR

MAP_REAL_TO_INT := rToLow;

// equality test made here is to prevent division by 0
IF rFromHigh <> rFromLow THEN
   MAP_REAL_TO_INT := TO_INT((rValue - rFromLow) * (rToHigh - rToLow) / (rFromHigh - rFromLow) + rToLow + 0.5);
END_IF

END_FUNCTION

// ---- POUs/20_AUTO/ST100/F_GetPercent_2.TcPOU
FUNCTION F_GetPercent_2 : INT
VAR_INPUT
    iAktStep      : INT; // actual step
    iStepP1_start : INT; // step process 1 start
    iStepP1_stop  : INT; // step process 1 stop
    iStepP2_start : INT; // step process 2 start
    iStepP2_stop  : INT; // step process 2 stop
END_VAR
VAR
END_VAR


IF iAktStep < iStepP1_start THEN
    F_GetPercent_2 := 0;

ELSIF iAktStep > iStepP1_stop AND iAktStep < iStepP2_start THEN
    F_GetPercent_2 := 50;

ELSIF iAktStep > iStepP2_stop THEN
    F_GetPercent_2 := 100;

ELSIF iAktStep >= iStepP1_start AND iAktStep <= iStepP1_stop THEN
    F_GetPercent_2 := 50 * (iAktStep - iStepP1_start) / ((iStepP1_stop - iStepP1_start) + 1);

ELSIF iAktStep >= iStepP2_start AND iAktStep <= iStepP2_stop THEN
    F_GetPercent_2 := 50 + 50 * (iAktStep - iStepP2_start) / ((iStepP2_stop - iStepP2_start) + 1);

ELSE
    F_GetPercent_2 := 0;

END_IF

END_FUNCTION

// ---- POUs/20_AUTO/ST105/FB_ABL_105_Feeder.TcPOU
FUNCTION_BLOCK FB_ABL_105_Feeder
(****************************************************************************************)
(*	TITEL				RFID-Ring laden, Feeder and rotary table                        *)
(*	Status				ungetestet                         								*)
(*	Beschrieb:			Ablaufbeschreibung												*)
(*																						*)
(*	Steps:	self-explained using enum													*)
(***********************************Revisionen*******************************************)
(*	see github blames																	*)
(****************************************************************************************)

VAR_INPUT
    xIN_Reset       : BOOL;          // Schrittkette zurücksetzen 
    xIN_Init        : BOOL;          // Initialisieren
    xIN_Quit        : BOOL;          // Fehler quittieren 
    xIN_Start       : BOOL;          // Startbefehl
    xIN_Sperre      : BOOL;          // FB Sperren 
    xIN_NextStep    : BOOL;          // Nächsten Schritt ausführen 
    xIN_AlarmAktiv  : BOOL;          // Anlage hat Alarm
    xIN_DryCycle    : BOOL;          // Fahren ohne Teile
    xIN_RestartCYCL : BOOL;          // Zyklus erneut starten im STEP, END, LEERFAHREN
    enIN_State      : enState;       // Status Anlage
    tIN_Timeout     : TIME := T#10s; // Timout

    pxFG_Freigabe : POINTER TO BOOL; //Freigabe von Station

    // Application specific
    xIN_PickPiece : BOOL; (* signal from the pick and place element
                             the number of picked signal depend on the recipe *)
    xIN_RotTableBlockedByPnp : BOOL; // Is the pick and place blocking the rotary table?
END_VAR
VAR_OUTPUT
    (* standart Ausgänge *)
    xOUT_ErrFlag  : BOOL;           // Error Flag 
    xOUT_Busy     : BOOL;           // Baustein befindet sich im Ablauf 
    xOUT_Done     : BOOL;           // Baustein hat den Ablauf beendet 		
    xOUT_Ready    : BOOL;           // Ready to begin, should be the same state as done	
    xOUT_Timeout  : BOOL;           // Timeout FB 
    xOUT_InitDone : BOOL;           // initialisierung fertig
    xOUT_Wait     : BOOL;           // Wartet auf Bedingung
    iOUT_Step     : ST105_Feeder_e; // Aktueller Schritt 
    sOUT_Step     : STRING;         // Aktueller Schritt but in string format
    bOUT_Error    : BYTE;           // Fehlernummer

    // Application specific
    xOUT_PceReadyToPick : BOOL; // the piece(s) is/are ready to picked
END_VAR
VAR
    (* Standard *)
    (* Schritt *)
    iLastStep : ST105_Feeder_e; // Merker letzter Schritt 
    iPreStep  : ST105_Feeder_e; // Schritt zurück nach Alarm 
    iAktStep  : ST105_Feeder_e; // aktueller Schritt

    // Trigger Starten 
    rtSTART : R_TRIG;
    // Timer TimeOut 
    TON_Timeout : TON;

    (* Bausteine *)

    // Application specific
    fb_axis105_10W               : FB_AxisLMturn_V1_1;
    simu_axis105_10W             : FB_Simu_AxisLM_V1_1;
    fb_feeder_wf                 : FB_Feeder2Sensors;
    fifo                         : FB_Fifo(4);
    simu_feeder                  : FB_Simu_Feeder; // simulation of a feeder
    simu_fifo_feeder_to_rotTable : FB_Fifo(20);    // fifo to hold a piece
    simu_fifo_feeder_lf          : FB_Fifo(20);    // fifo to hold a piece
    rtPutPiece                   : R_TRIG;         // trigger to add a piece
    fb_feeder_lf                 : FB_Feeder2Sensors;

    rtPick : R_TRIG; // r_trig signal from the pick and place machine

    iCurrentTableIndex : INT; // current table index
    iSearchIndex       : INT; (* Initialization index TO see how many element we have AT startup
                                 or after an alarm *)

    rDegreeToNextSlot : REAL; // how many degree is needed to rotate to the next slot

    eSliderStep    : ST105_Slider_e := ST105_Slider_e.slider_pusher_in;
    ton_two_pieces : TON; // TON for the detection of a piece inside one another

    fb_slider   : FB_ZylMo2El_V2_1;
    simu_slider : FB_Simu_Zyl2Pos;
    fb_pusher   : FB_ZylMo2El_V2_1;
    simu_pusher : FB_Simu_Zyl2Pos;

END_VAR
VAR CONSTANT
    MAX_SEARCH_TURN : INT := 4; // maximum search number

    FEEDER_SIMULATION : BOOL := FALSE; // Simulate this code
END_VAR

(*******************************************************************)
(* Trigger  *)
(*******************************************************************)
(* Zurücksetzen *)
IF xIN_RESET THEN
    iPreStep    := ST105_Feeder_e.RESET;
    iOUT_Step   := ST105_Feeder_e.RESET;
    eSliderStep := ST105_Slider_e.slider_pusher_in;
END_IF;

(* Error Quittieren *)
IF (bOUT_Error <> 0) AND xIN_Quit THEN
    xOUT_ErrFlag := FALSE;
    bOUT_Error   := 0;
    iOUT_Step    := iPreStep;
    eSliderStep  := ST105_Slider_e.slider_pusher_in;
END_IF;

iCurrentTableIndex := iCurrentTableIndex MOD 3;

IF _20_AUTO.recipe.st105.FeederSize <> 0 THEN
    rDegreeToNextSlot := REAL#360.0 / DINT_TO_REAL(_20_AUTO.recipe.st105.FeederSize);
ELSE
    rDegreeToNextSlot := REAL#90.0;
END_IF

(*******************************************************************)
(* Timer *)
(*******************************************************************)
TON_Timeout(IN := xIN_NextStep AND (iLastStep = iOUT_Step) (*todo FG *) ,
            PT := tIN_Timeout);

ton_two_pieces(IN := IO_BOX.I8705_ST105_Kontrolle_zwei_Filtergehiluse,
               PT := T#300MS);

(*******************************************************************)
(* Bausteine *)
(*******************************************************************)

fb_feeder_wf(xIN_Enable                := enIN_State = enState.StateAUTO OR enIN_State = enState.StateSTEP,
             xIN_PieceInEnd            := IO_BOX.I8600_ST105_teil_in_vereinzelung,
             xIN_PieceMax              := IO_BOX.I8600_ST105_teil_in_vereinzelung,
             xIN_InSimulation          := FEEDER_SIMULATION AND CONST.USE_SIMULATION,
             refIN_SimulatedFifo       := simu_fifo_feeder_to_rotTable,
             iIN_FifoSetMaxSensorValue := 10,
             diIN_SignlFilter_ms       := 500,
             diIN_StartDelay_ms        := 0,
             diIN_StopDelay_ms         := 10000,
             diIN_EmptyDelay_ms        := 0);

fb_feeder_lf(xIN_Enable                := enIN_State = enState.StateAUTO OR enIN_State = enState.StateSTEP,
             xIN_PieceInEnd            := IO_BOX.I8704_ST105_Maximum_LF,
             xIN_PieceMax              := IO_BOX.I8704_ST105_Maximum_LF,
             xIN_InSimulation          := FEEDER_SIMULATION AND CONST.USE_SIMULATION,
             refIN_SimulatedFifo       := simu_fifo_feeder_lf,
             iIN_FifoSetMaxSensorValue := 10,
             diIN_SignlFilter_ms       := _20_AUTO.recipe.st105.FeederConfig.InFilterDelay,
             diIN_StartDelay_ms        := _20_AUTO.recipe.st105.FeederConfig.StartDelay,
             diIN_StopDelay_ms         := _20_AUTO.recipe.st105.FeederConfig.StopDelay,
             diIN_EmptyDelay_ms        := _20_AUTO.recipe.st105.FeederConfig.EmptyDelay);

simu_feeder(xIN_Enable         := fb_feeder_wf.xOUT_EnableFeeder AND FEEDER_SIMULATION AND CONST.USE_SIMULATION,
            xIN_PceSensor      := fb_feeder_wf.xIN_PieceInEnd,
            tIN_NewPieceTime   := 500,
            iIN_WaitTimeMin_ms := 500,
            iIN_WaitTimeMax_ms := 1000);

rtPick(CLK := xIN_PickPiece);
rtPutPiece(CLK := simu_feeder.xOUT_NewPiece);

IF rtPutPiece.Q AND NOT simu_fifo_feeder_to_rotTable.IsFull() THEN
    simu_fifo_feeder_to_rotTable.Put(1);
END_IF

IF ST105_Feeder_e.Init_simu_home_table = iOUT_Step THEN
    fb_axis105_10W.rIN_Position :=
        TO_REAL(rDegreeToNextSlot - LMOD(ST105_Axis.axis105_10W.rActPos, rDegreeToNextSlot));

ELSIF ST105_Feeder_e.Init_apply_feeder_offset = iOUT_Step THEN
    fb_axis105_10W.rIN_Position := _20_AUTO.recipe.st105.RotaryTableOffset;

ELSE
    fb_axis105_10W.rIN_Position := rDegreeToNextSlot;

END_IF

simu_axis105_10W(xIN_Enable          := FEEDER_SIMULATION AND CONST.USE_SIMULATION,
                 wIN_AxisState       := ST105_Axis.axis105_10W.wState,
                 bIN_AxisCntr        := fb_axis105_10W.bOUT_AxisCntr,
                 udiIN_HomingTime_ms := 1000,
                 pIN_axisSimu        := ADR(SIMU.axis_ref[Axis_e.ST105_10W]),
                 pIN_axisHW          := ADR(ST105_Axis.axis105_10W.axis),
                 rIN_PosActual       := fb_axis105_10W.rOUT_ActPos,
                 rIN_PosMax          := ST105_Axis.const105_10W.POS_MAX,
                 rIN_PosMin          := ST105_Axis.const105_10W.POS_MIN,
                 rIN_PixMax          := 0,
                 rIN_PixMin          := 0);

fb_axis105_10W(enIN_State     := enIN_State,
               parIN_Buttons  := ADR(AXIS.btTeachArAxis[Axis_e.ST105_10W]),
               xIN_DisButtons := FALSE,
               xIN_Quit       := xIN_Quit,
               xIN_PARAMok    := TRUE,
               xIN_FREE       := NOT xIN_RotTableBlockedByPnp,
               xIN_FREE_HOME  := TRUE,
               rIN_POSMIN     := ST105_Axis.const105_10W.POS_MIN,
               rIN_POSMAX     := ST105_Axis.const105_10W.POS_MAX,
               rIN_VELOMAX    := ST105_Axis.const105_10W.VELO_MAX,
               rIN_VELOMANU   := ST105_Axis.const105_10W.VELO_MANU,
               rIN_VELOOPEN   := ST105_Axis.const105_10W.VELO_MANU / 4,
               rIN_JogInc     := AXIS.rTeachIncAxis,
               xIN_Execute    := ST105_Feeder_e.Init_set_table_pos = iOUT_Step OR
                                 ST105_Feeder_e.Init_table_go_to_zero = iOUT_Step OR
                                 ST105_Feeder_e.Init_simu_home_table = iOUT_Step OR
                                 ST105_Feeder_e.load_piece = iOUT_Step OR
                                 ST105_Feeder_e.Init_apply_feeder_offset = iOUT_Step,
               xIN_Relative     := fb_axis105_10W.xIN_Execute,
               xIN_STOP         := FALSE,
               xIN_OFF          := FALSE,
               rIN_Position     :=, // Is set above
               rIN_Velocity     := TO_REAL(100.0),
               rIN_Acceleration := TO_REAL(1440.0),
               rIN_Deceleration := TO_REAL(1440.0),
               rIN_Jerk         := TO_REAL(720000.0),
               rIN_PosManu      := TO_REAL(_20_AUTO.recipe.linearAxis[LinearAxis_e.ST105_11Z]
                                               .movesList[AXIS.bTeachPos[Axis_e.ST105_11Z]].lrPosition),
               xIN_Home  := ST105_feeder_e.Init_home_table = iOUT_Step,
               xIN_Reset := xIN_Reset OR ST105_feeder_e.RESET = iOUT_Step,
               // The simu fb gives us the hardware signal when we are not in simulation
               wAxisState    := simu_axis105_10W.wOUT_AxisState,
               bOUT_AxisCntr => ST105_Axis.axis105_10W.bCtrlHi,
               rOUT_ActPos   =>, // leave empty, rActPos must be set using the modulo
               axisIN_REF    := simu_axis105_10W.pOUT_axisRef^);

ST105_Axis.axis105_10W.rActPos := LREAL_TO_REAL(simu_axis105_10W.pOUT_axisRef^.NcToPlc.ModuloActPos);

// pneumatics
fb_slider(xIN_Reset    := xIN_Reset OR (ST105_Feeder_e.RESET = iOUT_Step),
          xIN_Quit     := xIN_Quit,
          xIN_Manu     := enState.StateMANU = enIN_State,
          pbtIN_Button := ADR(HMI.btManuCylinders[StationList_e.ST105][1]),
          xIN_GS       := simu_slider.xOUT_inGS,
          xIN_AS       := simu_slider.xOUT_inAS,
          xIN_FREE     := TRUE,
          xINtoGS      := ST105_Slider_e.slider_go_down = eSliderStep,
          xINtoAS      := ST105_Slider_e.slider_go_up = eSliderStep,
          tIN_ErrAS    := DINT_TO_TIME(_20_AUTO.recipe.cylinder2Pos[StationList_e.ST105]
                                           [ST105_Cylinders_e.Ausschieber_ab_auf].toAS_alarm_time),
          tIN_ErrGS := DINT_TO_TIME(_20_AUTO.recipe.cylinder2Pos[StationList_e.ST105]
                                        [ST105_Cylinders_e.Ausschieber_ab_auf].toGS_alarm_time),
          tIN_WaitAS := DINT_TO_TIME(_20_AUTO.recipe.cylinder2Pos[StationList_e.ST105]
                                         [ST105_Cylinders_e.Ausschieber_ab_auf].toAS_wait_time),
          tIN_WaitGS := DINT_TO_TIME(_20_AUTO.recipe.cylinder2Pos[StationList_e.ST105]
                                         [ST105_Cylinders_e.Ausschieber_ab_auf].toGS_wait_time));

simu_slider(xIN_Enable := FEEDER_SIMULATION AND CONST.USE_SIMULATION,
            xIN_inGS   := IO_BOX.I8700_ST105_Ausheber_unten_GS,
            xIN_inAS   := IO_BOX.I8701_ST105_Ausheber_oben_AS,
            xIN_valve  := fb_slider.xOUT_VALVE,
            tIN_GS_ms  := 200,  //ms
            tIN_AS_ms  := 200); //ms

fb_pusher(xIN_Reset    := xIN_Reset OR (ST105_Feeder_e.RESET = iOUT_Step),
          xIN_Quit     := xIN_Quit,
          xIN_Manu     := enState.StateMANU = enIN_State,
          pbtIN_Button := ADR(HMI.btManuCylinders[StationList_e.ST105][2]),
          xIN_GS       := simu_pusher.xOUT_inGS,
          xIN_AS       := simu_pusher.xOUT_inAS,
          xIN_FREE     := TRUE,
          xINtoGS      := ST105_Slider_e.slider_pusher_in = eSliderStep,
          xINtoAS      := ST105_Slider_e.slider_push_out = eSliderStep,
          tIN_ErrAS    := DINT_TO_TIME(_20_AUTO.recipe.cylinder2Pos[StationList_e.ST105]
                                           [ST105_Cylinders_e.Ausschieber_ab_auf].toAS_alarm_time),
          tIN_ErrGS := DINT_TO_TIME(_20_AUTO.recipe.cylinder2Pos[StationList_e.ST105]
                                        [ST105_Cylinders_e.Ausschieber_ab_auf].toGS_alarm_time),
          tIN_WaitAS := DINT_TO_TIME(_20_AUTO.recipe.cylinder2Pos[StationList_e.ST105]
                                         [ST105_Cylinders_e.Ausschieber_ab_auf].toAS_wait_time),
          tIN_WaitGS := DINT_TO_TIME(_20_AUTO.recipe.cylinder2Pos[StationList_e.ST105]
                                         [ST105_Cylinders_e.Ausschieber_ab_auf].toGS_wait_time));

simu_pusher(xIN_Enable := FEEDER_SIMULATION AND CONST.USE_SIMULATION,
            xIN_inGS   := IO_BOX.I8702_ST105_Abschieber_zuruck_GS,
            xIN_inAS   := IO_BOX.I8703_ST105_Abschieber_vor_AS,
            xIN_valve  := fb_pusher.xOUT_VALVE,
            tIN_GS_ms  := 200,  //ms
            tIN_AS_ms  := 200); //ms

(*******************************************************************)
(* OUTPUTS *)
(*******************************************************************)
// Error Flag 
xOUT_ErrFlag := (bOUT_Error <> 0) OR (ST105_Feeder_e.ERROR = iOUT_Step);
// Baustein befindet sich im Ablauf 
xOUT_Busy := (iOUT_Step > ST105_Feeder_e.READY) AND (iOUT_Step < ST105_Feeder_e.DONE);
// Baustein hat den Ablauf beendet
xOUT_Done := (iOUT_Step = ST105_Feeder_e.DONE);
// Process ready
xOUT_Ready := (iOUT_Step = ST105_Feeder_e.READY);
// Timeout FB 				 		
xOUT_Timeout := TON_Timeout.Q;
// Itialisierung fertig			
xOUT_InitDone := (iOUT_Step = ST105_Feeder_e.READY);
// Aktueller Schritt			
iOUT_Step := iOUT_Step; //Im Ablauf gesetzt		
sOUT_Step := TO_STRING(iOUT_Step);
//Fehlernummer	 
bOUT_Error := bOUT_Error; //Im Ablauf/FB gesetzt	
(* Warte (alle Schritte wo auf FG oder Teile gewartet wird) *)
xOUT_Wait := (iOUT_Step = ST105_Feeder_e.DONE) OR
             (iOUT_Step = ST105_Feeder_e.READY);

IO_BOX.Q9500_ST105_Freigabe_WF := fb_feeder_wf.xOUT_EnableFeeder AND
                                  NOT (FEEDER_SIMULATION AND CONST.USE_SIMULATION) AND
                                  ((ST105_Slider_e.slider_down = eSliderStep) OR
                                  ((ST105_Slider_e.slider_go_up = eSliderStep) AND fb_slider.xIN_GS));

IO_BOX.Q9501_ST105_Freigabe_LF := fb_feeder_lf.xOUT_EnableFeeder AND
                                  IO_BOX.Q9500_ST105_Freigabe_WF AND
                                  NOT (FEEDER_SIMULATION AND CONST.USE_SIMULATION) AND
                                  (ST105_Slider_e.slider_down = eSliderStep);

OUT.Q106_ST105_zusatz_band_on := IO_BOX.Q9501_ST105_Freigabe_LF;

IO_BOX.Q8800_14_Auschieber_ab_auf :=
    fb_slider.xOUT_VALVE AND NOT (FEEDER_SIMULATION AND CONST.USE_SIMULATION);

IO_BOX.Q8801_14_Auschieber_vor_zuruck :=
    fb_pusher.xOUT_VALVE AND NOT (FEEDER_SIMULATION AND CONST.USE_SIMULATION);

xOUT_PceReadyToPick := ST105_Feeder_e.DONE = iOUT_Step;

(*******************************************************************)
(* Ablauf *)
(*******************************************************************)

(* Sperren *)
IF xIN_Sperre THEN
    iPreStep    := ST105_Feeder_e.RESET;
    iOUT_Step   := ST105_Feeder_e.RESET;
    eSliderStep := ST105_Slider_e.slider_pusher_in;
    RETURN;
END_IF;

(* Schritt Merker *)
IF iAktStep <> iOUT_Step THEN
    iLastStep := iAktStep;
    iAktStep  := iOUT_Step;
END_IF

(* START *)
rtSTART(CLK := xIN_Start);

IF 0 = bOUT_Error THEN
    IF fb_axis105_10W.xOUT_ErrFlag THEN
        bOUT_Error := 11;
    ELSIF fb_slider.xOUT_ErrFlag THEN
        bOUT_Error := 12;
    ELSIF fb_pusher.xOUT_ErrFlag THEN
        bOUT_Error := 13;
    END_IF
ELSIF iOUT_Step < ST105_Feeder_e.ERROR THEN
    iOUT_Step := ST105_Feeder_e.ERROR;
END_IF

(*******************************************************************)
(* Schrittkette slider tower *)
(*******************************************************************)
CASE eSliderStep OF
ST105_Slider_e.slider_down:
    IF xIN_NextStep AND ton_two_pieces.Q AND enIN_State >= enState.StateAUTO THEN
        eSliderStep := ST105_Slider_e.slider_go_up;
    END_IF

ST105_Slider_e.slider_go_up:
    IF xIN_NextStep AND fb_slider.xOUT_inAS THEN
        eSliderStep := ST105_Slider_e.slider_push_out;
    END_IF

ST105_Slider_e.slider_push_out:
    IF xIN_NextStep AND fb_pusher.xOUT_inAS THEN
        eSliderStep := ST105_Slider_e.slider_pusher_in;
    END_IF

ST105_Slider_e.slider_pusher_in:
    IF xIN_NextStep AND fb_pusher.xOUT_inGS THEN
        eSliderStep := ST105_Slider_e.slider_go_down;
    END_IF

ST105_Slider_e.slider_go_down:
    IF xIN_NextStep AND fb_slider.xOUT_inGS THEN
        eSliderStep := ST105_Slider_e.slider_down;
    END_IF

END_CASE

(*******************************************************************)
(* Schrittkette  *)
(*******************************************************************)
CASE iOUT_Step OF

(***** RESET *****)
ST105_Feeder_e.RESET: (* Schritt 0-99 *)
    //Initialisierungen
    //Start Init Ablauf
    IF xIN_Init THEN
        iOUT_Step := ST105_Feeder_e.INIT;
        //Start Manu Ablauf
    ELSIF enIN_State = StateMANU AND xIN_NextStep THEN
        iOUT_Step := ST105_Feeder_e.INIT;
    END_IF;

(***** INIT *****)
ST105_Feeder_e.INIT: (* Grundstellung ? *)
    IF NOT xIN_RotTableBlockedByPnp THEN
        iOUT_Step := ST105_Feeder_e.Init_home_table;
    END_IF

ST105_Feeder_e.Init_home_table:
    IF fb_axis105_10W.xOUT_HOMED THEN
        iCurrentTableIndex := 0;
		iOUT_Step := ST105_Feeder_e.Init_apply_feeder_offset;
    END_IF

ST105_Feeder_e.Init_apply_feeder_offset:
    IF fb_axis105_10W.xOUT_DONE THEN
        IF FEEDER_SIMULATION AND CONST.USE_SIMULATION THEN
            iOUT_Step := ST105_Feeder_e.Init_simu_home_table;
        ELSE
            iOUT_Step := ST105_Feeder_e.Init_reset_search_index;
        END_IF
    END_IF

ST105_Feeder_e.Init_simu_home_table:
    IF fb_axis105_10W.xOUT_DONE THEN
        iOUT_Step := ST105_Feeder_e.Init_reset_search_index;
    END_IF

ST105_Feeder_e.Init_table_go_to_zero:
    IF fb_axis105_10W.xOUT_DONE THEN
        iOUT_Step := ST105_Feeder_e.Init_reset_search_index;
    END_IF

ST105_Feeder_e.Init_reset_search_index:
    iSearchIndex := 0;
    fifo.Empty();
    iOUT_Step := ST105_Feeder_e.READY; // bypass unusefull search cycle

ST105_Feeder_e.Init_set_table_pos:
    IF fb_axis105_10W.xOUT_DONE THEN
        iCurrentTableIndex := iCurrentTableIndex + 1;
        iOUT_Step          := ST105_Feeder_e.Init_see_if_piece_there;
    END_IF

ST105_Feeder_e.Init_see_if_piece_there:
    IF simu_feeder.xOUT_NewPiece THEN
        fifo.Put(1);
    END_IF

    IF iSearchIndex < MAX_SEARCH_TURN THEN
        iOUT_Step    := ST105_Feeder_e.Init_set_table_pos;
        iSearchIndex := iSearchIndex + 1;
    ELSE
        iOUT_Step := ST105_Feeder_e.READY;
    END_IF

(***** READY / INIT DONE *****)
ST105_Feeder_e.READY: (* Start AUTO,END,LEER,STEP *)
    IF xIN_Start THEN //IF rtSTART.Q THEN
        iOUT_Step := ST105_Feeder_e.START;
    END_IF

(***** START  ZYKLISCH *****)
ST105_Feeder_e.START: (*  *)
    IF xIN_NextStep AND pxFG_Freigabe^ THEN
        iOUT_Step := ST105_Feeder_e.check_if_feeding_necessary;
        iPreStep  := ST105_Feeder_e.READY;
    END_IF;

ST105_Feeder_e.check_if_feeding_necessary:
    IF (fifo.GetLen() >= _20_AUTO.recipe.st105.FeederSize) OR fifo.IsFull() THEN
        iOUT_Step := ST105_Feeder_e.DONE;
    ELSE
        iOUT_Step := ST105_Feeder_e.wait_on_a_piece;
    END_IF

ST105_Feeder_e.wait_on_a_piece:
    IF (FEEDER_SIMULATION AND CONST.USE_SIMULATION AND NOT simu_fifo_feeder_to_rotTable.IsEmpty()) OR
       (NOT (FEEDER_SIMULATION AND CONST.USE_SIMULATION) AND IO_BOX.I8600_ST105_teil_in_vereinzelung) THEN
        iOUT_Step := ST105_Feeder_e.load_piece;
        simu_fifo_feeder_to_rotTable.Pop(1);
    END_IF

ST105_Feeder_e.load_piece:
    IF fb_axis105_10W.xOUT_DONE THEN
        fifo.Put(1);
        iOUT_Step := ST105_Feeder_e.check_if_feeding_necessary;
    END_IF

(***** DONE *****)
ST105_Feeder_e.DONE: (* Letzter Schritt  *)
    IF rtPick.Q THEN
        fifo.Pop(TO_INT(_20_AUTO.recipe.st105.xUseVerLeft));
        fifo.Pop(TO_INT(_20_AUTO.recipe.st105.xUseVerRight));
    END_IF

    IF NOT xIN_AlarmAktiv THEN
        //AUTO
        IF (enIN_State = StateAUTO) AND xIN_RestartCYCL AND (fifo.GetLen() < _20_AUTO.recipe.st105.FeederSize)
            THEN
            iOUT_Step := ST105_Feeder_e.START;
            // We don't load pieces when not in auto

            //STEP / END / LEERFAHREN fertig
        ELSIF (enIN_State = StateREADY) THEN
            iOUT_Step := ST105_Feeder_e.READY;
        END_IF;
    END_IF;

(************ ERROR *************)
ST105_Feeder_e.ERROR: (* ERROR *) ;

END_CASE;

END_FUNCTION_BLOCK

// ---- POUs/20_AUTO/Simu/FB_Simu_Feeder.TcPOU
// This simu FB is used to generate pieces randomly
// A piece is given during a given amount of time throug 'xOUT_NewPiece'
// Use this output as your nearest sensor 
FUNCTION_BLOCK FB_Simu_Feeder
VAR_INPUT
    xIN_Enable         : BOOL; // enable the feeder
    tIN_NewPieceTime   : DINT;
    iIN_WaitTimeMin_ms : DINT;
    iIN_WaitTimeMax_ms : DINT;
END_VAR
VAR_OUTPUT
    xOUT_NewPiece : BOOL;
END_VAR
VAR
    _rand          : DRAND;
    _enableClock   : BOOL  := FALSE;
    _startTime_ms  : UDINT := 0;
    _timeToWait_ms : DINT := 0;
END_VAR

IF xIN_Enable AND NOT _EnableClock THEN
    THIS^.GetNewRandomTime();
    xOUT_NewPiece := FALSE;
END_IF

_EnableClock := xIN_Enable;

IF xIN_Enable AND THIS^.IsTimeElapsed() THEN
    IF NOT xOUT_NewPiece THEN
        _timeToWait_ms := tIN_NewPieceTime;
		THIS^._startTime_ms := GetTick();
    ELSE
        THIS^.GetNewRandomTime();
    END_IF

    xOUT_NewPiece := NOT xOUT_NewPiece;
ELSIF NOT xIN_Enable THEN
    xOUT_NewPiece := FALSE;
END_IF

METHOD FB_init : BOOL
VAR_INPUT
	bInitRetains : BOOL; // if TRUE, the retain variables are initialized (warm start / cold start)
	bInCopyCode : BOOL;  // if TRUE, the instance afterwards gets moved into the copy code (online change)
END_VAR
VAR
END_VAR
this^._rand.Seed := TO_INT(F_GetSystemTime());
END_METHOD

METHOD PRIVATE GetNewRandomTime : BOOL
VAR_INPUT
END_VAR
THIS^._startTime_ms := GetTick();
THIS^._rand();
THIS^._timeToWait_ms :=
    TO_DINT(THIS^._rand.Num * (THIS^.iIN_WaitTimeMax_ms - THIS^.iIN_WaitTimeMin_ms) + THIS^.iIN_WaitTimeMin_ms);
END_METHOD

METHOD IsTimeElapsed : BOOL
VAR_INPUT
END_VAR
IsTimeElapsed := TO_DINT(GetTick() - _startTime_ms) > _timeToWait_ms;
END_METHOD

END_FUNCTION_BLOCK

// ---- POUs/20_AUTO/Simu/FB_Simu_Zyl2Pos.TcPOU
// Simu fb for FB_ZylMo2El_V2_1
FUNCTION_BLOCK FB_Simu_Zyl2Pos
VAR_INPUT
    xIN_Enable : BOOL; // enable this FB. You should only enable this FB when you are sure to be in sumulation modes
    xIN_inGS   : BOOL; // connect to the sensor inGS
    xIN_inAS   : BOOL; // connect to the sensor inAS
    xIN_valve  : BOOL; // connect to valve output of the simulated valve
    tIN_GS_ms  : DINT; // time in ms when GS signal should be on
    tIN_AS_ms  : DINT; // time in ms when AS signal should be on
END_VAR
VAR_OUTPUT
    xOUT_inGS : BOOL; // in GS position 
    xOUT_inAS : BOOL; // in AS position 
END_VAR
VAR
    _tick       : UDINT;
    _in_gs_tick : UDINT;
    _in_as_tick : UDINT;
END_VAR

_tick := GetTick();

IF xIN_valve THEN
    _in_gs_tick := _tick;
END_IF

IF NOT xIN_valve THEN
    _in_as_tick := _tick;
END_IF

xOUT_inGS := xIN_Enable AND (TO_LINT(_tick - _in_gs_tick) > tIN_GS_ms) OR
             NOT xIN_Enable AND xIN_inGS;

xOUT_inAS := xIN_Enable AND (TO_LINT(_tick - _in_as_tick) > tIN_AS_ms) OR
             NOT xIN_Enable AND xIN_inAS;

END_FUNCTION_BLOCK

// ---- POUs/20_AUTO/ST110/FB_AUT_110.TcPOU
FUNCTION_BLOCK FB_AUT_110 EXTENDS FB_AUT_ABSTRACT
(****************************************************************************)
(*	POU_AUT_zxx			Bausteinaufrufe Station	zxx							*)
(*	Status				ungetestet											*)
(*  Version:			1.0													*)
(*	Beschrieb:																*)
(*																			*)
(*	Abläufe:			FB_ABLzxxA		Hauptablauf							*)
(*																			*)
(*																			*)
(* 	25.09.2019/Dj															*)
(****************************************************************************)
(*	dd.mm.yyyy   KZ    x.y			Beschrieb								*)
(****************************************************************************)
VAR_INPUT
    (* spezifische Eingänge *)

END_VAR
VAR_OUTPUT
    (* spezifische Ausgänge *)

END_VAR
VAR
    (* Bausteine *)
    fb_Pnp    : FB_ABL_110_Pnp;
    fb_Feeder : FB_ABL_110_Feeder;

    fb_stat_pnp    : FB_AUT_Statistics;
    fb_stat_Feeder : FB_AUT_Statistics;

END_VAR

VAR CONSTANT
    ROT_TABLE_FREE_MAX_Y : REAL := 100.0; // If Y and Z axis is more than this value, the feeder cannot move
    ROT_TABLE_FREE_MAX_Z : REAL := 50.0;  // If Z and Y axis is more than this value, the feeder cannot move
END_VAR

(*******************************************************************)
(* Timer *)
(*******************************************************************)

(*******************************************************************)
(* Flanken / Merker *)
(*******************************************************************)
//MANU CYCLE
IF (enIN_State = StateMANU) AND xIN_ManuCycle THEN
    xManuCycle := TRUE;
END_IF;

IF (enIN_State <> StateMANU) OR xOUT_Done THEN
    xManuCycle := FALSE;
END_IF

//NEXT STEP
xNextStep := (enIN_State > StateSTEP) OR
             ((enIN_State = StateSTEP) AND xIN_Step) OR
             ((enIN_State = StateMANU) AND xManuCycle);

//RESET
xReset := (enIN_State < StateREADY) AND (enIN_State <> StateINIT) AND NOT xManuCycle;

(*******************************************************************)
(* Bausteinaufrufe Abläufe *)
(*******************************************************************)

xRelease := MAIN.MoverMan.IsProcessUsed(THIS^);

fb_Pnp(xIN_Reset          := xReset,
       xIN_Init           := xIN_Init,
       xIN_Quit           := xIN_Quit,
       xIN_Start          := enIN_State >= enState.StateLEER AND xRelease,
       xIN_Sperre         := NOT xIN_On,
       xIN_NextStep       := xNextStep,
       xIN_AlarmAktiv     := xIN_AlarmAktiv,
       xIN_DryCycle       := xIN_DryCycle,
       xIN_RestartCYCL    := enIN_State >= enState.StateLEER,
       enIN_State         := enIN_State,
       tIN_Timeout        := tIN_Timeout,
       pxFG_Freigabe      := ADR(xRelease),
       Mover              := THIS^.Mover,
       xIN_PceReadyToPick := fb_Feeder.xOUT_Done);

fb_Feeder(xIN_Reset       := xReset,
          xIN_Init        := xIN_Init,
          xIN_Quit        := xIN_Quit,
          xIN_Start       := enIN_State >= enState.StateLEER AND xRelease,
          xIN_Sperre      := NOT xIN_On,
          xIN_NextStep    := xNextStep,
          xIN_AlarmAktiv  := xIN_AlarmAktiv,
          xIN_DryCycle    := xIN_DryCycle,
          xIN_RestartCYCL := enIN_State >= enState.StateLEER,
          enIN_State      := enIN_State,
          tIN_Timeout     := tIN_Timeout,
          pxFG_Freigabe   := ADR(xRelease),
          // special
          xIN_PickPiece            := fb_Pnp.xOUT_PickPiece,
          xIN_RotTableBlockedByPnp := (ST110_Axis.axis110_01Y.rActPos > ROT_TABLE_FREE_MAX_Y) AND
                                      (ST110_Axis.axis110_02Z.rActPos > ROT_TABLE_FREE_MAX_Z));

fb_stat_pnp(xIN_Enable  := enState.StateAUTO = enIN_State,
            xIN_Waiting := fb_Pnp.xOUT_Wait,
            xIN_Running := (fb_Pnp.iOUT_Step >= ST110_Pnp_e.START) AND
                           (fb_Pnp.iOUT_Step <= ST110_Pnp_e.DONE),
            // Since we use a mover system, a cycle is done when we are waiting on a mover
            xIN_Done := fb_Pnp.iOUT_Step = ST110_Pnp_e.waitOnMover);

fb_stat_Feeder(xIN_Enable  := enState.StateAUTO = enIN_State,
               xIN_Waiting := fb_feeder.xOUT_Wait,
               xIN_Running := (fb_feeder.iOUT_Step >= ST110_Feeder_e.START) AND
                              (fb_feeder.iOUT_Step <= ST110_Feeder_e.DONE),
               xIN_Done := fb_feeder.iOUT_Step = ST110_Feeder_e.DONE);

(*******************************************************************)
(* Mover reset flags *)
(*******************************************************************)

(*******************************************************************)
(* OUTPUT *)
(*******************************************************************)
xOUT_InitDone := fb_Pnp.xOUT_InitDone AND fb_Feeder.xOUT_InitDone;
xOUT_Ready    := fb_Pnp.xOUT_Ready AND fb_Feeder.xOUT_Ready;
xOUT_Done     := fb_Pnp.xOUT_Done;
xOUT_ErrFlag  := fb_Pnp.xOUT_ErrFlag OR fb_Feeder.xOUT_ErrFlag;
xOUT_Wait     := fb_Pnp.xOUT_Wait AND fb_Feeder.xOUT_Wait;
xOUT_AlarmST  := xOUT_ErrFlag;

IF fb_Pnp.xOUT_ErrFlag THEN
    bOUT_ErrorNum := fb_Pnp.bOUT_Error;
ELSIF fb_Feeder.xOUT_ErrFlag THEN
    bOUT_ErrorNum := fb_Feeder.bOUT_Error;
ELSE
	bOUT_ErrorNum := 0;
END_IF

(*******************************************************************)
(* Bausteinaufruf Error Station *)
(*******************************************************************)
POU_ALARM_110(xIN_QUIT      := xIN_Quit,
              iIN_ArraySize := ST110_Alarm_e._max,
              pstrIN_ALARM  := ADR(HMI.strArALARM[21]),
              refPOU        := THIS^);

(* % of completion of the process *)
PROPERTY iCompletionPC : INT
GET
iCompletionPC := THIS^.fb_Pnp.iOUT_ProcessCompletion;
END_GET
END_PROPERTY

PROPERTY ProcessExecution : ProcessExecution_e
GET
ProcessExecution := THIS^._ProcessExecution;
END_GET
SET
THIS^._ProcessExecution := ProcessExecution;
END_SET
END_PROPERTY

PROPERTY xBusy : BOOL
GET
xBusy := THIS^.fb_Pnp.xOUT_Busy;
END_GET
SET
END_SET
END_PROPERTY

PROPERTY xDone : BOOL
GET
xDone := THIS^.fb_Pnp.xOUT_Ready OR THIS^.fb_Pnp.xOUT_Done;
END_GET
END_PROPERTY

PROPERTY xMoverPathFree : BOOL
GET
xMoverPathFree := THIS^.fb_Pnp.xOUT_MoverFree OR THIS^.fb_Pnp.xOUT_Ready OR THIS^.fb_Pnp.xOUT_Done;
END_GET
END_PROPERTY

PROPERTY xMoverShouldLeave : BOOL
GET
xMoverShouldLeave := THIS^.fb_Pnp.iOUT_Step = ST110_Pnp_e.SYNC_MOVER_LEAVE;
END_GET
END_PROPERTY

END_FUNCTION_BLOCK

// ---- POUs/20_AUTO/ST110/FB_ABL_110_Pnp.TcPOU
FUNCTION_BLOCK FB_ABL_110_Pnp
(****************************************************************************************)
(*	TITEL				RFID-Ring laden		    										*)
(*	Status				ungetestet                         								*)
(*	Beschrieb:			Ablaufbeschreibung												*)
(*																						*)
(*	Steps:	self-explained using enum													*)
(***********************************Revisionen*******************************************)
(*	see github blames																	*)
(****************************************************************************************)

VAR_INPUT
    xIN_Reset       : BOOL;          // Schrittkette zurücksetzen 
    xIN_Init        : BOOL;          // Initialisieren
    xIN_Quit        : BOOL;          // Fehler quittieren 
    xIN_Start       : BOOL;          // Startbefehl
    xIN_Sperre      : BOOL;          // FB Sperren 
    xIN_NextStep    : BOOL;          // Nächsten Schritt ausführen 
    xIN_AlarmAktiv  : BOOL;          // Anlage hat Alarm
    xIN_DryCycle    : BOOL;          // Fahren ohne Teile
    xIN_RestartCYCL : BOOL;          // Zyklus erneut starten im STEP, END, LEERFAHREN
    enIN_State      : enState;       // Status Anlage
    tIN_Timeout     : TIME := T#10s; // Timout

    pxFG_Freigabe : POINTER TO BOOL; //Freigabe von Station

    // Application specific
    Mover              : REFERENCE TO FB_Mover;
    xIN_PceReadyToPick : BOOL; // the piece(s) is/are ready to picked
END_VAR
VAR_OUTPUT
    (* standart Ausgänge *)
    xOUT_ErrFlag  : BOOL;        // Error Flag 
    xOUT_Busy     : BOOL;        // Baustein befindet sich im Ablauf 
    xOUT_Done     : BOOL;        // Baustein hat den Ablauf beendet 		
    xOUT_Ready    : BOOL;        // Ready to begin, should be the same state as done	
    xOUT_Timeout  : BOOL;        // Timeout FB 
    xOUT_InitDone : BOOL;        // initialisierung fertig
    xOUT_Wait     : BOOL;        // Wartet auf Bedingung
    iOUT_Step     : ST110_Pnp_e; // Aktueller Schritt 
    sOUT_Step     : STRING;      // Aktueller Schritt but in string format
    bOUT_Error    : BYTE;        // Fehlernummer

    iOUT_ProcessCompletion : INT;  //process completion, express in % (0-100)
    xOUT_MoverFree         : BOOL; // The mover is free to move
    xOUT_PickPiece         : BOOL; // Set to true when a piece is picked

END_VAR
VAR
    (* Standard *)
    (* Schritt *)
    iLastStep : ST110_Pnp_e; // Merker letzter Schritt 
    iPreStep  : ST110_Pnp_e; // Schritt zurück nach Alarm 
    iAktStep  : ST110_Pnp_e; // aktueller Schritt

    // Trigger Starten 
    rtSTART : R_TRIG;
    // Timer TimeOut 
    TON_Timeout : TON;

    (* Bausteine *)

    (* Spezial *)
    fb_axis110_01Y : FB_AxisLM_V1_1;
    fb_axis110_02Z : FB_AxisLIN_V1_1;
    fb_axis110_03Z : FB_AxisLIN_V1_1;
    fb_axis110_04Z : FB_AxisLIN_V1_1;

    fb_PnpHorAxis  : FB_LinearMotionMan;
    fb_PnpVerAxisL : FB_LinearMotionMan;
    fb_PnpVerAxisR : FB_LinearMotionMan;
    fb_PnpVerAxisU : FB_LinearMotionMan;

    fb_simu_axis110_01Y : FB_Simu_AxisLM_V1_1;
    fb_simu_axis110_02Z : FB_Simu_AxisLIN_V1_1;
    fb_simu_axis110_03Z : FB_Simu_AxisLIN_V1_1;
    fb_simu_axis110_04Z : FB_Simu_AxisLIN_V1_1;

    fb_gripperLeft    : FB_ZylMo2El_V2_1;
    simu_gripperLeft  : FB_Simu_Zyl2Pos;
    fb_gripperRight   : FB_ZylMo2El_V2_1;
    simu_gripperRight : FB_Simu_Zyl2Pos;

    fb_kraftLeft  : FB_WandlerForceSensor;
    fb_kraftRight : FB_WandlerForceSensor;
	
	xIsPiecesPicked : BOOL; // Do we have pieces picked by vacum

END_VAR
VAR CONSTANT
    PNP_SIMULATION       : BOOL := FALSE; // Set to TRUE to simulate this part of the program
    PNP_DONT_CHECK_KRAFT : BOOL := FALSE; // don't care of kraft sensor
END_VAR

(*******************************************************************)
(* Trigger  *)
(*******************************************************************)
(* Zurücksetzen *)
IF xIN_RESET THEN
    iPreStep  := ST110_Pnp_e.RESET;
    iOUT_Step := ST110_Pnp_e.RESET;
END_IF;

(* Error Quittieren *)
IF (bOUT_Error <> 0) AND xIN_Quit THEN
    xOUT_ErrFlag := FALSE;
    bOUT_Error   := 0;
    iOUT_Step    := iPreStep;
END_IF;

(*******************************************************************)
(* Timer *)
(*******************************************************************)
TON_Timeout(IN := xIN_NextStep AND (iLastStep = iOUT_Step) (*todo FG *) ,
            PT := tIN_Timeout);

(*******************************************************************)
(* Bausteine *)
(*******************************************************************)
fb_PnpHorAxis(config          := _20_AUTO.recipe.linearAxis[LinearAxis_e.ST110_01Y],
              xIN_Init        := enIN_State = enState.StateINIT,
              xIN_Reset       := xIN_Reset,
              lrIN_CurrPos    := fb_axis110_01Y.rOUT_ActPos,
              lrIN_Delta_mm   := 0.5,
              iIN_CurrentStep := iOUT_Step,
              iIN_moveNumber  := ST110_PnpHorPos_e._max);

fb_simu_axis110_01Y(xIN_Enable          := PNP_SIMULATION AND CONST.USE_SIMULATION,
                    bIN_AxisCntr        := fb_axis110_01Y.bOUT_AxisCntr,
                    wIN_AxisState       := ST110_Axis.axis110_01Y.wState,
                    udiIN_HomingTime_ms := 2000,
                    pIN_axisSimu        := ADR(SIMU.axis_ref[Axis_e.ST110_01Y]),
                    pIN_axisHW          := ADR(ST110_Axis.axis110_01Y.axis),
                    rIN_PosActual       := fb_axis110_01Y.rOUT_ActPos,
                    rIN_PosMax          := ST110_Axis.const110_01Y.POS_MAX,
                    rIN_PosMin          := ST110_Axis.const110_01Y.POS_MIN,
                    rIN_PixMax          := 100,
                    rIN_PixMin          := 0);

fb_axis110_01Y(enIN_State       := enIN_State,
               parIN_Buttons    := ADR(AXIS.btTeachArAxis[Axis_e.ST110_01Y]),
               xIN_DisButtons   :=,
               xIN_Quit         := xIN_Quit,
               xIN_PARAMok      := TRUE, (*TODO*)
               xIN_FREE         := TRUE,
               xIN_FREE_HOME    := TRUE,
               rIN_POSMIN       := ST110_Axis.const110_01Y.POS_MIN,
               rIN_POSMAX       := ST110_Axis.const110_01Y.POS_MAX,
               rIN_VELOMAX      := ST110_Axis.const110_01Y.VELO_MAX,
               rIN_VELOMANU     := ST110_Axis.const110_01Y.VELO_MANU,
               rIN_VELOOPEN     := ST110_Axis.const110_01Y.VELO_MANU / 4,
               rIN_JogInc       := AXIS.rTeachIncAxis,
               xIN_Execute      := fb_PnpHorAxis.xOUT_Execute,
               xIN_Home         := ST110_Pnp_e.Init_HomeHorizontals = iOUT_Step,
               xIN_Relative     :=,
               rIN_Position     := TO_REAL(fb_PnpHorAxis.OUT_MoveProfile.lrPosition),
               rIN_Velocity     := TO_REAL(fb_PnpHorAxis.OUT_MoveProfile.lrVelocity),
               rIN_Acceleration := TO_REAL(fb_PnpHorAxis.OUT_MoveProfile.lrAccel),
               rIN_Deceleration := TO_REAL(fb_PnpHorAxis.OUT_MoveProfile.lrDecel),
               rIN_Jerk         := TO_REAL(fb_PnpHorAxis.OUT_MoveProfile.lrJerk),
               rIN_PosManu      := TO_REAL(_20_AUTO.recipe.linearAxis[LinearAxis_e.ST110_01Y]
                                               .movesList[AXIS.bTeachPos[Axis_e.ST110_01Y]].lrPosition),
               rIN_VeloJogManu := TO_REAL(Axis.rJogVelo_pc),
               xIN_Reset       := (ST110_Pnp_e.RESET = iOUT_Step) OR xIN_Reset,
               // the simu fb gives the hardware signal when not in simulation
               wAxisState    := fb_simu_axis110_01Y.wOUT_AxisState,
               rOUT_ActPos   => ST110_Axis.axis110_01Y.rActPos,
               bOUT_AxisCntr => ST110_Axis.axis110_01Y.bCtrlHi,
               axisIN_REF    := fb_simu_axis110_01Y.pOUT_axisRef^);

fb_PnpVerAxisL(config          := _20_AUTO.recipe.linearAxis[LinearAxis_e.ST110_02Z],
               xIN_Init        := enIN_State = enState.StateINIT,
               xIN_Reset       := xIN_Reset,
               lrIN_CurrPos    := fb_axis110_02Z.rOUT_ActPos,
               lrIN_Delta_mm   := 0.05,
               iIN_CurrentStep := iOUT_Step,
               iIN_moveNumber  := ST110_PnpVerPos_e._max);

fb_simu_axis110_02Z(xIN_InSimu    := PNP_SIMULATION AND CONST.USE_SIMULATION,
                    rIN_PosActual := fb_axis110_02Z.rOUT_ActPos,
                    pIN_axisSimu  := ADR(SIMU.axis_ref[Axis_e.ST110_02Z]),
                    pIN_axisHW    := ADR(ST110_Axis.axis110_02Z.axis),
                    rIN_PosMax    := ST110_Axis.const110_02Z.POS_MAX,
                    rIN_PosMin    := ST110_Axis.const110_02Z.POS_MIN,
                    rIN_PixMax    := 80,
                    rIN_PixMin    := 0);

fb_axis110_02Z(enIN_State     := enIN_State,
               parIN_Buttons  := ADR(AXIS.btTeachArAxis[Axis_e.ST110_02Z]),
               xIN_DisButtons :=,
               xIN_Quit       := xIN_Quit,
               xIN_AX5000     := TRUE,
               xIN_ENC_ABS    := TRUE, // TODO set accordingly
               xIN_PARAMok    := TRUE,
               xIN_FREE       := TRUE,
               xIN_Halt       := NOT ((ST110_Pnp_e.PnP_Ver_ShuttleTorqueControl = iOUT_Step) AND
                                 fb_kraftRight.lrOUT_value >= _20_AUTO.recipe.st110.kraft_right_raw) AND
                                 NOT (ST110_Pnp_e.PnP_Ver_quick_stop = iOUT_Step),
               xIN_FREE_HOME   := TRUE,
               rIN_POSMIN      := ST110_Axis.const110_02Z.POS_MIN,
               rIN_POSMAX      := ST110_Axis.const110_02Z.POS_MAX,
               rIN_VELOMAX     := ST110_Axis.const110_02Z.VELO_MAX,
               rIN_VELOMANU    := ST110_Axis.const110_02Z.VELO_MANU,
               rIN_VELOOPEN    := ST110_Axis.const110_02Z.POS_MAX / 4,
               rIN_JogInc      := AXIS.rTeachIncAxis,
               rIN_VeloJogManu := TO_REAL(AXIS.rJogVelo_pc),
               xIN_HomeExe     :=,
               xIN_HomeCalib   :=,
               xIN_Execute     := (_20_AUTO.recipe.st110.xUseVerLeft OR (iOUT_Step < ST110_Pnp_e.READY)) AND
                                  (fb_PnpVerAxisL.xOUT_Execute),
               xIN_HomeExe      :=,
               xIN_Relative     :=,
               rIN_Position     := TO_REAL(fb_PnpVerAxisL.OUT_MoveProfile.lrPosition),
               rIN_Velocity     := TO_REAL(fb_PnpVerAxisL.OUT_MoveProfile.lrVelocity),
               rIN_Acceleration := TO_REAL(fb_PnpVerAxisL.OUT_MoveProfile.lrAccel),
               rIN_Deceleration := TO_REAL(fb_PnpVerAxisL.OUT_MoveProfile.lrDecel),
               rIN_Jerk         := TO_REAL(fb_PnpVerAxisL.OUT_MoveProfile.lrJerk),
               rIN_PosManu      := TO_REAL(_20_AUTO.recipe.linearAxis[LinearAxis_e.ST110_02Z]
                                               .movesList[AXIS.bTeachPos[Axis_e.ST110_02Z]].lrPosition),
               xIN_Reset := (ST110_Pnp_e.RESET = iOUT_Step) OR xIN_Reset,
               // output
               rOUT_ActPos => ST110_Axis.axis110_02Z.rActPos,
               axisIN_REF  := fb_simu_axis110_02Z.pOUT_axisRef^);

fb_PnpVerAxisR(config          := _20_AUTO.recipe.linearAxis[LinearAxis_e.ST110_03Z],
               xIN_Init        := enIN_State = enState.StateINIT,
               xIN_Reset       := xIN_Reset,
               lrIN_CurrPos    := fb_axis110_03Z.rOUT_ActPos,
               lrIN_Delta_mm   := 0.05,
               iIN_CurrentStep := iOUT_Step,
               iIN_moveNumber  := ST110_PnpVerPos_e._max);

fb_simu_axis110_03Z(xIN_InSimu    := PNP_SIMULATION AND CONST.USE_SIMULATION,
                    rIN_PosActual := fb_axis110_03Z.rOUT_ActPos,
                    pIN_axisSimu  := ADR(SIMU.axis_ref[Axis_e.ST110_03Z]),
                    pIN_axisHW    := ADR(ST110_Axis.axis110_03Z.axis),
                    rIN_PosMax    := ST110_Axis.const110_03Z.POS_MAX,
                    rIN_PosMin    := ST110_Axis.const110_03Z.POS_MIN,
                    rIN_PixMax    := 80,
                    rIN_PixMin    := 0);

fb_axis110_03Z(enIN_State     := enIN_State,
               parIN_Buttons  := ADR(AXIS.btTeachArAxis[Axis_e.ST110_03Z]),
               xIN_DisButtons :=,
               xIN_Quit       := xIN_Quit,
               xIN_PARAMok    := TRUE, (*TODO*)
               xIN_FREE       := TRUE,
               xIN_Halt       := NOT ((ST110_Pnp_e.PnP_Ver_ShuttleTorqueControl = iOUT_Step) AND
                                 fb_kraftRight.lrOUT_value >= _20_AUTO.recipe.st110.kraft_right_raw) AND
                                 NOT (ST110_Pnp_e.PnP_Ver_quick_stop = iOUT_Step),
               xIN_FREE_HOME := TRUE,
               rIN_POSMIN    := ST110_Axis.const110_03Z.POS_MIN,
               rIN_POSMAX    := ST110_Axis.const110_03Z.POS_MAX,
               rIN_VELOMAX   := ST110_Axis.const110_03Z.VELO_MAX,
               rIN_VELOMANU  := ST110_Axis.const110_03Z.VELO_MANU,
               rIN_VELOOPEN  := ST110_Axis.const110_03Z.VELO_MANU / 4,
               rIN_JogInc    := AXIS.rTeachIncAxis,
               xIN_Execute   := (_20_AUTO.recipe.st110.xUseVerRight OR (iOUT_Step < ST110_Pnp_e.READY)) AND
                                (fb_PnpVerAxisR.xOUT_Execute),
               xIN_HomeExe      :=,
               xIN_Relative     :=,
               rIN_Position     := TO_REAL(fb_PnpVerAxisR.OUT_MoveProfile.lrPosition),
               rIN_Velocity     := TO_REAL(fb_PnpVerAxisR.OUT_MoveProfile.lrVelocity),
               rIN_Acceleration := TO_REAL(fb_PnpVerAxisR.OUT_MoveProfile.lrAccel),
               rIN_Deceleration := TO_REAL(fb_PnpVerAxisR.OUT_MoveProfile.lrDecel),
               rIN_Jerk         := TO_REAL(fb_PnpVerAxisR.OUT_MoveProfile.lrJerk),
               rIN_PosManu      :=
               TO_REAL(_20_AUTO.recipe
                           .linearAxis[LinearAxis_e.ST110_03Z].movesList[AXIS.bTeachPos[Axis_e.ST110_03Z]].lrPosition),
               xIN_Reset   := (ST110_Pnp_e.RESET = iOUT_Step) OR xIN_Reset,
               axisIN_REF  := fb_simu_axis110_03Z.pOUT_axisRef^,
               xIN_AX5000  := TRUE,
               xIN_ENC_ABS := TRUE,
               rOUT_ActPos => ST110_Axis.axis110_03Z.rActPos,
               axisIN_REF  := fb_simu_axis110_03Z.pOUT_axisRef^);

fb_PnpVerAxisU(config          := _20_AUTO.recipe.linearAxis[LinearAxis_e.ST110_04Z],
               xIN_Init        := enState.StateINIT = enIN_State,
               xIN_Reset       := xIN_Reset,
               lrIN_CurrPos    := ST110_Axis.axis110_04Z.rActPos,
               lrIN_Delta_mm   := 0.5,
               iIN_CurrentStep := iOUT_Step,
               iIN_moveNumber  := ST110_PnpVerPushPos_e._max);

fb_simu_axis110_04Z(xIN_InSimu    := PNP_SIMULATION AND CONST.USE_SIMULATION,
                    rIN_PosActual := ST110_Axis.axis110_04Z.rActPos,
                    pIN_axisSimu  := ADR(SIMU.axis_ref[Axis_e.ST110_04Z]),
                    pIN_axisHW    := ADR(ST110_Axis.axis110_04Z.axis),
                    rIN_PosMax    := ST110_Axis.const110_04Z.POS_MAX,
                    rIN_PosMin    := ST110_Axis.const110_04Z.POS_MIN,
                    rIN_PixMax    := 80,
                    rIN_PixMin    := 0);

